IF (PVL.s8098[s8098_mapping.FT_202].PDO.VolumeFlow.Status.eStatus=burkert.eSensor_Status.Low_Low_Alarm)	THEN	tStatus:=ez202_Status.FT202_Low_Low_Flow_Alarm;		END_IF;
IF (PVL.s8098[s8098_mapping.FT_202].PDO.VolumeFlow.Status.eStatus=burkert.eSensor_Status.HiHi_Alarm)	THEN	tStatus:=ez202_Status.FT202_High_High_Flow_Alarm;		END_IF;
IF (PVL.s8098[s8098_mapping.FT_203].PDO.VolumeFlow.Status.eStatus=burkert.eSensor_Status.Low_Low_Alarm)	THEN	tStatus:=ez202_Status.FT203_Low_Low_Flow_Alarm;		END_IF;
IF (PVL.s8098[s8098_mapping.FT_203].PDO.VolumeFlow.Status.eStatus=burkert.eSensor_Status.HiHi_Alarm)	THEN	tStatus:=ez202_Status.FT202_High_High_Flow_Alarm;		END_IF;


IF PVl.s8312[s8312_mapping.PT_202].Status.eStatus= Burkert.eSensor_Status.HiHi_Alarm THEN tStatus:=eZ202_Status.PT202_High_Pressure_Alarm; END_IF;
IF PVl.s8312[s8312_mapping.PT_202].Status.eStatus= Burkert.eSensor_Status.Low_Low_Alarm THEN tStatus:=eZ202_Status.PT202_Low_Pressure_Alarm; END_IF;
///////********		IF PVl.s8312[s8312_mapping.PT_203].Status.eStatus= Burkert.eSensor_Status.HiHi_Alarm THEN tStatus:=eZ202_Status.PT203_High_Pressure_Alarm; END_IF;
///////********		IF PVl.s8312[s8312_mapping.PT_203].Status.eStatus= Burkert.eSensor_Status.Low_Low_Alarm THEN tStatus:=eZ202_Status.PT203_Low_Pressure_Alarm; END_IF;

Test_ALL:=tStatus;
                
END_METHOD

METHOD Test_Drain_P202 : eZ202_Status
  VAR_INPUT
    Status : eZ202_status;
  END_VAR
  VAR
    tStatus : eZ202_Status;
  END_VAR
                  tStatus:=Status;
IF NOT(GVL.Filter_Path_Available) THEN tStatus:=eZ202_Status.No_Filter_Available; END_IF;

//IF NOT(GVL.s3363[s3363_mapping.ACV_203].Ready) 	THEN 	tStatus:=eZ202_Status.ACV203_Not_Ready; 	END_IF;
//IF NOT(GVL.s3363[s3363_mapping.ACV_206].Ready) 	THEN 	tStatus:=eZ202_Status.ACV206_Not_Ready; 	END_IF;
//IF NOT(GVL.s3363[s3363_mapping.ACV_224].Ready) 	THEN 	tStatus:=eZ202_Status.ACV224_Not_Ready; 	END_IF;
//IF NOT(GVL.s3363[s3363_mapping.ACV_225].Ready) 	THEN 	tStatus:=eZ202_Status.ACV225_Not_Ready; 	END_IF;
IF NOT(GVL.s3363[s3363_mapping.ACV_226].Ready) 	THEN 	tStatus:=eZ202_Status.ACV226_Not_Ready; 	END_IF;
IF NOT(Network.VFD[VFD_Mapping.VFD_202].Ready) 	THEN	tStatus:=eZ202_status.P202_Not_Ready;		END_IF;
//IF NOT(Network.VFD[VFD_Mapping.VFD_203].Ready) 	THEN	tStatus:=eZ202_status.P203_Not_Ready;		END_IF;
IF NOT(PVL.Ait[AIT_Mapping.LT_202].Ready) 		THEN	tStatus:=eZ202_Status.LT202_Not_Ready;		END_IF;
//IF NOT(PVL.Ait[AIT_Mapping.LT_202A].Ready) 		THEN	tStatus:=eZ202_Status.LT202A_Not_Ready;		END_IF;
IF NOT(PVl.s8312[s8312_mapping.PT_202].Ready)	THEN	tStatus:=ez202_Status.PT202_Not_Ready;		END_IF;
//IF NOT(PVl.s8312[s8312_mapping.PT_203].Ready)	THEN	tStatus:=ez202_Status.PT203_Not_Ready;		END_IF;
IF NOT(PVL.s8098[s8098_mapping.FT_202].Ready)	THEN	tStatus:=ez202_Status.FT202_Not_Ready;		END_IF;
//IF NOT(PVL.s8098[s8098_mapping.FT_203].Ready)	THEN	tStatus:=ez202_Status.FT203_Not_Ready;		END_IF;
IF gvl.LS[ls_mapping.LSLL_205].Status.eStatus=Burkert.DI_Status.No_Liquid_Detected_Alarm	THEN	tStatus:=eZ202_Status.Drain_Complete;		END_IF;
//IF gvl.LS[ls_mapping.LSLL_203].Status.eStatus=Burkert.DI_Status.No_Liquid_Detected_Alarm	THEN	tStatus:=eZ202_Status.P203_Intake_Empty;		END_IF;
//IF gvl.LS[ls_mapping.LSHH_201].Status.eStatus=Burkert.DI_Status.Liquid_Detected_Alarm		THEN	tStatus:=eZ202_Status.EP101_High_High_Alarm;	END_IF;
//IF (PVL.Ait[AIT_Mapping.LT_202].Ready) 		THEN	tStatus:=eZ202_Status.LT202_Not_Ready;		END_IF;
//IF (PVL.Ait[AIT_Mapping.LT_202A].Ready) 		THEN	tStatus:=eZ202_Status.LT202A_Not_Ready;		END_IF;
//IF GVL.s3363[s3363_mapping.ACV_203].Status.eStatus=Burkert.eACV_Status.Pos_Error THEN	tStatus:=eZ202_Status.ACV203_Error; END_IF;
//IF GVL.s3363[s3363_mapping.ACV_206].Status.eStatus=Burkert.eACV_Status.Pos_Error THEN	tStatus:=eZ202_Status.ACV206_Error; END_IF;
//IF GVL.s3363[s3363_mapping.ACV_224].Status.eStatus=Burkert.eACV_Status.Pos_Error THEN	tStatus:=eZ202_Status.ACV224_Error; END_IF;
//IF GVL.s3363[s3363_mapping.ACV_225].Status.eStatus=Burkert.eACV_Status.Pos_Error THEN	tStatus:=eZ202_Status.ACV225_Error; END_IF;
IF GVL.s3363[s3363_mapping.ACV_226].Status.eStatus=Burkert.eACV_Status.Pos_Error THEN	tStatus:=eZ202_Status.ACV226_Error; END_IF;
//IF PVL.AIT[AIT_Mapping.LT_202].Status.eStatus=Burkert.eSensor_Status.Low_Low_Alarm THEN	tStatus:=eZ202_Status.LT202_Low_Low_Alarm;	END_IF;
//IF PVL.AIT[AIT_Mapping.LT_202A].Status.eStatus=Burkert.eSensor_Status.Low_Low_Alarm THEN	tStatus:=eZ202_Status.LT202A_Low_Low_Alarm;	END_IF;
IF (PVL.s8098[s8098_mapping.FT_202].PDO.VolumeFlow.Status.eStatus=burkert.eSensor_Status.Low_Low_Alarm)	THEN	tStatus:=ez202_Status.FT202_Low_Low_Flow_Alarm;		END_IF;
//IF (PVL.s8098[s8098_mapping.FT_202].PDO.VolumeFlow.Status.eStatus=burkert.eSensor_Status.HiHi_Alarm)	THEN	tStatus:=ez202_Status.FT202_High_High_Flow_Alarm;		END_IF;
//IF (PVL.s8098[s8098_mapping.FT_203].PDO.VolumeFlow.Status.eStatus=burkert.eSensor_Status.Low_Low_Alarm)	THEN	tStatus:=ez202_Status.FT203_Low_Low_Flow_Alarm;		END_IF;
//IF (PVL.s8098[s8098_mapping.FT_203].PDO.VolumeFlow.Status.eStatus=burkert.eSensor_Status.HiHi_Alarm)	THEN	tStatus:=ez202_Status.FT202_High_High_Flow_Alarm;		END_IF;
IF PVl.s8312[s8312_mapping.PT_202].Status.eStatus= Burkert.eSensor_Status.HiHi_Alarm THEN tStatus:=eZ202_Status.PT202_High_Pressure_Alarm; END_IF;
IF PVl.s8312[s8312_mapping.PT_202].Status.eStatus= Burkert.eSensor_Status.Low_Low_Alarm THEN tStatus:=eZ202_Status.PT202_Low_Pressure_Alarm; END_IF;
//IF PVl.s8312[s8312_mapping.PT_203].Status.eStatus= Burkert.eSensor_Status.HiHi_Alarm THEN tStatus:=eZ202_Status.PT203_High_Pressure_Alarm; END_IF;
//IF PVl.s8312[s8312_mapping.PT_203].Status.eStatus= Burkert.eSensor_Status.Low_Low_Alarm THEN tStatus:=eZ202_Status.PT203_Low_Pressure_Alarm; END_IF;

Test_Drain_P202:=tStatus;
                
END_METHOD

METHOD Test_Drain_P203 : eZ202_Status
  VAR_INPUT
    Status : eZ202_status;
  END_VAR
  VAR
    tStatus : eZ202_Status;
  END_VAR
                  tStatus:=Status;
IF NOT(GVL.Filter_Path_Available) THEN tStatus:=eZ202_Status.No_Filter_Available; END_IF;

//IF NOT(GVL.s3363[s3363_mapping.ACV_203].Ready) 	THEN 	tStatus:=eZ202_Status.ACV203_Not_Ready; 	END_IF;
//IF NOT(GVL.s3363[s3363_mapping.ACV_206].Ready) 	THEN 	tStatus:=eZ202_Status.ACV206_Not_Ready; 	END_IF;
//IF NOT(GVL.s3363[s3363_mapping.ACV_224].Ready) 	THEN 	tStatus:=eZ202_Status.ACV224_Not_Ready; 	END_IF;
//IF NOT(GVL.s3363[s3363_mapping.ACV_225].Ready) 	THEN 	tStatus:=eZ202_Status.ACV225_Not_Ready; 	END_IF;
IF NOT(GVL.s3363[s3363_mapping.ACV_226].Ready) 	THEN 	tStatus:=eZ202_Status.ACV226_Not_Ready; 	END_IF;
IF NOT(Network.VFD[VFD_Mapping.VFD_202].Ready) 	THEN	tStatus:=eZ202_status.P202_Not_Ready;		END_IF;
//IF NOT(Network.VFD[VFD_Mapping.VFD_203].Ready) 	THEN	tStatus:=eZ202_status.P203_Not_Ready;		END_IF;
IF NOT(PVL.Ait[AIT_Mapping.LT_202].Ready) 		THEN	tStatus:=eZ202_Status.LT202_Not_Ready;		END_IF;
//IF NOT(PVL.Ait[AIT_Mapping.LT_202A].Ready) 		THEN	tStatus:=eZ202_Status.LT202A_Not_Ready;		END_IF;
IF NOT(PVl.s8312[s8312_mapping.PT_202].Ready)	THEN	tStatus:=ez202_Status.PT202_Not_Ready;		END_IF;
//IF NOT(PVl.s8312[s8312_mapping.PT_203].Ready)	THEN	tStatus:=ez202_Status.PT203_Not_Ready;		END_IF;
IF NOT(PVL.s8098[s8098_mapping.FT_202].Ready)	THEN	tStatus:=ez202_Status.FT202_Not_Ready;		END_IF;
//IF NOT(PVL.s8098[s8098_mapping.FT_203].Ready)	THEN	tStatus:=ez202_Status.FT203_Not_Ready;		END_IF;
//IF gvl.LS[ls_mapping.LSLL_205].Status.eStatus=Burkert.DI_Status.No_Liquid_Detected_Alarm	THEN	tStatus:=eZ202_Status.Drain_Complete;		END_IF;
IF gvl.LS[ls_mapping.LSLL_203].Status.eStatus=Burkert.DI_Status.No_Liquid_Detected_Alarm	THEN	tStatus:=eZ202_Status.Drain_Complete;		END_IF;
//IF gvl.LS[ls_mapping.LSHH_201].Status.eStatus=Burkert.DI_Status.Liquid_Detected_Alarm		THEN	tStatus:=eZ202_Status.EP101_High_High_Alarm;	END_IF;
//IF (PVL.Ait[AIT_Mapping.LT_202].Ready) 		THEN	tStatus:=eZ202_Status.LT202_Not_Ready;		END_IF;
//IF (PVL.Ait[AIT_Mapping.LT_202A].Ready) 		THEN	tStatus:=eZ202_Status.LT202A_Not_Ready;		END_IF;
//IF GVL.s3363[s3363_mapping.ACV_203].Status.eStatus=Burkert.eACV_Status.Pos_Error THEN	tStatus:=eZ202_Status.ACV203_Error; END_IF;
//IF GVL.s3363[s3363_mapping.ACV_206].Status.eStatus=Burkert.eACV_Status.Pos_Error THEN	tStatus:=eZ202_Status.ACV206_Error; END_IF;
//IF GVL.s3363[s3363_mapping.ACV_224].Status.eStatus=Burkert.eACV_Status.Pos_Error THEN	tStatus:=eZ202_Status.ACV224_Error; END_IF;
//IF GVL.s3363[s3363_mapping.ACV_225].Status.eStatus=Burkert.eACV_Status.Pos_Error THEN	tStatus:=eZ202_Status.ACV225_Error; END_IF;
IF GVL.s3363[s3363_mapping.ACV_226].Status.eStatus=Burkert.eACV_Status.Pos_Error THEN	tStatus:=eZ202_Status.ACV226_Error; END_IF;
//IF PVL.AIT[AIT_Mapping.LT_202].Status.eStatus=Burkert.eSensor_Status.Low_Low_Alarm THEN	tStatus:=eZ202_Status.LT202_Low_Low_Alarm;	END_IF;
//IF PVL.AIT[AIT_Mapping.LT_202A].Status.eStatus=Burkert.eSensor_Status.Low_Low_Alarm THEN	tStatus:=eZ202_Status.LT202A_Low_Low_Alarm;	END_IF;
IF (PVL.s8098[s8098_mapping.FT_202].PDO.VolumeFlow.Status.eStatus=burkert.eSensor_Status.Low_Low_Alarm)	THEN	tStatus:=ez202_Status.FT202_Low_Low_Flow_Alarm;		END_IF;
//IF (PVL.s8098[s8098_mapping.FT_202].PDO.VolumeFlow.Status.eStatus=burkert.eSensor_Status.HiHi_Alarm)	THEN	tStatus:=ez202_Status.FT202_High_High_Flow_Alarm;		END_IF;
//IF (PVL.s8098[s8098_mapping.FT_203].PDO.VolumeFlow.Status.eStatus=burkert.eSensor_Status.Low_Low_Alarm)	THEN	tStatus:=ez202_Status.FT203_Low_Low_Flow_Alarm;		END_IF;
//IF (PVL.s8098[s8098_mapping.FT_203].PDO.VolumeFlow.Status.eStatus=burkert.eSensor_Status.HiHi_Alarm)	THEN	tStatus:=ez202_Status.FT202_High_High_Flow_Alarm;		END_IF;
IF PVl.s8312[s8312_mapping.PT_202].Status.eStatus= Burkert.eSensor_Status.HiHi_Alarm THEN tStatus:=eZ202_Status.PT202_High_Pressure_Alarm; END_IF;
IF PVl.s8312[s8312_mapping.PT_202].Status.eStatus= Burkert.eSensor_Status.Low_Low_Alarm THEN tStatus:=eZ202_Status.PT202_Low_Pressure_Alarm; END_IF;
//IF PVl.s8312[s8312_mapping.PT_203].Status.eStatus= Burkert.eSensor_Status.HiHi_Alarm THEN tStatus:=eZ202_Status.PT203_High_Pressure_Alarm; END_IF;
//IF PVl.s8312[s8312_mapping.PT_203].Status.eStatus= Burkert.eSensor_Status.Low_Low_Alarm THEN tStatus:=eZ202_Status.PT203_Low_Pressure_Alarm; END_IF;

Test_Drain_P203:=tStatus;
                
END_METHOD

METHOD Test_Z201_Return_P202 : eZ202_Status
  VAR_INPUT
    Status : eZ202_status;
  END_VAR
  VAR
    tStatus : eZ202_Status;
  END_VAR
                  tStatus:=Status;


IF NOT(GVL.s3363[s3363_mapping.ACV_203].Ready) 	THEN 	tStatus:=eZ202_Status.ACV203_Not_Ready; 	END_IF;
IF NOT(GVL.s3363[s3363_mapping.ACV_206].Ready) 	THEN 	tStatus:=eZ202_Status.ACV206_Not_Ready; 	END_IF;
//IF NOT(GVL.s3363[s3363_mapping.ACV_224].Ready) 	THEN 	tStatus:=eZ202_Status.ACV224_Not_Ready; 	END_IF;
//IF NOT(GVL.s3363[s3363_mapping.ACV_225].Ready) 	THEN 	tStatus:=eZ202_Status.ACV225_Not_Ready; 	END_IF;
IF NOT(GVL.s3363[s3363_mapping.ACV_226].Ready) 	THEN 	tStatus:=eZ202_Status.ACV226_Not_Ready; 	END_IF;

IF NOT(Network.VFD[VFD_Mapping.VFD_202].Ready) 	THEN	tStatus:=eZ202_status.P202_Not_Ready;		END_IF;
//IF NOT(Network.VFD[VFD_Mapping.VFD_203].Ready) 	THEN	tStatus:=eZ202_status.P203_Not_Ready;		END_IF;

IF NOT(PVL.Ait[AIT_Mapping.LT_202].Ready) 		THEN	tStatus:=eZ202_Status.LT202_Not_Ready;		END_IF;
//IF NOT(PVL.Ait[AIT_Mapping.LT_202A].Ready) 		THEN	tStatus:=eZ202_Status.LT202A_Not_Ready;		END_IF;

///////********		IF NOT(PVl.s8312[s8312_mapping.PT_202].Ready)	THEN	tStatus:=ez202_Status.PT202_Not_Ready;		END_IF;
///////********		IF NOT(PVl.s8312[s8312_mapping.PT_203].Ready)	THEN	tStatus:=ez202_Status.PT203_Not_Ready;		END_IF;

//IF NOT(PVL.s8098[s8098_mapping.FT_202].Ready)	THEN	tStatus:=ez202_Status.FT202_Not_Ready;		END_IF;
//IF NOT(PVL.s8098[s8098_mapping.FT_203].Ready)	THEN	tStatus:=ez202_Status.FT203_Not_Ready;		END_IF;
	
IF gvl.LS[ls_mapping.LSLL_205].Status.eStatus=Burkert.DI_Status.No_Liquid_Detected_Alarm	THEN	tStatus:=eZ202_Status.P202_Intake_Empty;		END_IF;
//IF gvl.LS[ls_mapping.LSLL_203].Status.eStatus=Burkert.DI_Status.No_Liquid_Detected_Alarm	THEN	tStatus:=eZ202_Status.P203_Intake_Empty;		END_IF;
IF gvl.LS[ls_mapping.LSHH_201].Status.eStatus=Burkert.DI_Status.Liquid_Detected_Alarm		THEN	tStatus:=eZ202_Status.EP101_High_High_Alarm;	END_IF;

//IF NOT(PVL.Ait[AIT_Mapping.LT_202].Ready) 		THEN	tStatus:=eZ202_Status.LT202_Not_Ready;		END_IF;
//IF (PVL.Ait[AIT_Mapping.LT_202].Status.eStatus=Burkert.eSensor_Status.HiHi_Alarm) 		THEN	tStatus:=eZ202_Status.LT202_High_High_Alarm;		END_IF;

IF NOT(PVL.Ait[AIT_Mapping.LT_201].Ready) 		THEN	tStatus:=eZ202_Status.LT201_Not_Ready;		END_IF;
IF (PVL.Ait[AIT_Mapping.LT_201].Status.eStatus=Burkert.eSensor_Status.HiHi_Alarm) 		THEN	tStatus:=eZ202_Status.LT201_High_High_Alarm;		END_IF;

IF NOT(pVL.Ait[AIT_Mapping.LT_101_P].Ready) 		THEN	tStatus:=eZ202_Status.LT101_Not_Ready;		END_IF;
IF (PVL.Ait[AIT_Mapping.LT_101_P].Status.eStatus=Burkert.eSensor_Status.HiHi_Alarm) 		THEN	tStatus:=eZ202_Status.LT101_High_High_Alarm;		END_IF;

//IF (PVL.Ait[AIT_Mapping.LT_202A].Ready) 		THEN	tStatus:=eZ202_Status.LT202A_Not_Ready;		END_IF;


IF GVL.s3363[s3363_mapping.ACV_203].Status.eStatus=Burkert.eACV_Status.Pos_Error THEN	tStatus:=eZ202_Status.ACV203_Error; END_IF;
IF GVL.s3363[s3363_mapping.ACV_206].Status.eStatus=Burkert.eACV_Status.Pos_Error THEN	tStatus:=eZ202_Status.ACV206_Error; END_IF;
//IF GVL.s3363[s3363_mapping.ACV_224].Status.eStatus=Burkert.eACV_Status.Pos_Error THEN	tStatus:=eZ202_Status.ACV224_Error; END_IF;
//IF GVL.s3363[s3363_mapping.ACV_225].Status.eStatus=Burkert.eACV_Status.Pos_Error THEN	tStatus:=eZ202_Status.ACV225_Error; END_IF;
IF GVL.s3363[s3363_mapping.ACV_226].Status.eStatus=Burkert.eACV_Status.Pos_Error THEN	tStatus:=eZ202_Status.ACV226_Error; END_IF;

//IF NOT(GVL.Filter_Path_Available) THEN tStatus:=eZ202_Status.No_Filter_Available; END_IF;

//IF (PVL.s8098[s8098_mapping.FT_202].PDO.VolumeFlow.Status.eStatus=burkert.eSensor_Status.Low_Low_Alarm)	THEN	tStatus:=ez202_Status.FT202_Low_Low_Flow_Alarm;		END_IF;
//IF (PVL.s8098[s8098_mapping.FT_202].PDO.VolumeFlow.Status.eStatus=burkert.eSensor_Status.HiHi_Alarm)	THEN	tStatus:=ez202_Status.FT202_High_High_Flow_Alarm;		END_IF;
IF (PVL.s8098[s8098_mapping.FT_203].PDO.VolumeFlow.Status.eStatus=burkert.eSensor_Status.Low_Low_Alarm)	THEN	tStatus:=ez202_Status.FT203_Low_Low_Flow_Alarm;		END_IF;
//IF (PVL.s8098[s8098_mapping.FT_203].PDO.VolumeFlow.Status.eStatus=burkert.eSensor_Status.HiHi_Alarm)	THEN	tStatus:=ez202_Status.FT202_High_High_Flow_Alarm;		END_IF;


//IF PVl.s8312[s8312_mapping.PT_202].Status.eStatus= Burkert.eSensor_Status.HiHi_Alarm THEN tStatus:=eZ202_Status.PT202_High_Pressure_Alarm; END_IF;
//IF PVl.s8312[s8312_mapping.PT_202].Status.eStatus= Burkert.eSensor_Status.Low_Low_Alarm THEN tStatus:=eZ202_Status.PT202_Low_Pressure_Alarm; END_IF;
///////********		IF PVl.s8312[s8312_mapping.PT_203].Status.eStatus= Burkert.eSensor_Status.HiHi_Alarm THEN tStatus:=eZ202_Status.PT203_High_Pressure_Alarm; END_IF;
///////********		IF PVl.s8312[s8312_mapping.PT_203].Status.eStatus= Burkert.eSensor_Status.Low_Low_Alarm THEN tStatus:=eZ202_Status.PT203_Low_Pressure_Alarm; END_IF;

IF (PVL.Ait[AIT_Mapping.LT_202].Status.eStatus=Burkert.eSensor_Status.Low_Low_Alarm) 		THEN	tStatus:=eZ202_Status.LT202_Low_Low_Alarm;		END_IF;

Test_Z201_Return_P202:=tStatus;
                
END_METHOD

METHOD Test_Z201_Return_P203 : eZ202_Status
  VAR_INPUT
    Status : eZ202_status;
  END_VAR
  VAR
    tStatus : eZ202_Status;
  END_VAR
                  tStatus:=Status;


IF NOT(GVL.s3363[s3363_mapping.ACV_203].Ready) 	THEN 	tStatus:=eZ202_Status.ACV203_Not_Ready; 	END_IF;
//IF NOT(GVL.s3363[s3363_mapping.ACV_206].Ready) 	THEN 	tStatus:=eZ202_Status.ACV206_Not_Ready; 	END_IF;
//IF NOT(GVL.s3363[s3363_mapping.ACV_224].Ready) 	THEN 	tStatus:=eZ202_Status.ACV224_Not_Ready; 	END_IF;
//IF NOT(GVL.s3363[s3363_mapping.ACV_225].Ready) 	THEN 	tStatus:=eZ202_Status.ACV225_Not_Ready; 	END_IF;
IF NOT(GVL.s3363[s3363_mapping.ACV_226].Ready) 	THEN 	tStatus:=eZ202_Status.ACV226_Not_Ready; 	END_IF;

//IF NOT(Network.VFD[VFD_Mapping.VFD_202].Ready) 	THEN	tStatus:=eZ202_status.P202_Not_Ready;		END_IF;
IF NOT(Network.VFD[VFD_Mapping.VFD_203].Ready) 	THEN	tStatus:=eZ202_status.P203_Not_Ready;		END_IF;

IF NOT(PVL.Ait[AIT_Mapping.LT_202].Ready) 		THEN	tStatus:=eZ202_Status.LT202_Not_Ready;		END_IF;
//IF NOT(PVL.Ait[AIT_Mapping.LT_202A].Ready) 		THEN	tStatus:=eZ202_Status.LT202A_Not_Ready;		END_IF;

//IF NOT(PVl.s8312[s8312_mapping.PT_202].Ready)	THEN	tStatus:=ez202_Status.PT202_Not_Ready;		END_IF;
///////********		IF NOT(PVl.s8312[s8312_mapping.PT_203].Ready)	THEN	tStatus:=ez202_Status.PT203_Not_Ready;		END_IF;

//IF NOT(PVL.s8098[s8098_mapping.FT_202].Ready)	THEN	tStatus:=ez202_Status.FT202_Not_Ready;		END_IF;
//IF NOT(PVL.s8098[s8098_mapping.FT_203].Ready)	THEN	tStatus:=ez202_Status.FT203_Not_Ready;		END_IF;
	
//IF gvl.LS[ls_mapping.LSLL_205].Status.eStatus=Burkert.DI_Status.No_Liquid_Detected_Alarm	THEN	tStatus:=eZ202_Status.P202_Intake_Empty;		END_IF;
IF gvl.LS[ls_mapping.LSLL_203].Status.eStatus=Burkert.DI_Status.No_Liquid_Detected_Alarm	THEN	tStatus:=eZ202_Status.P203_Intake_Empty;		END_IF;
IF gvl.LS[ls_mapping.LSHH_201].Status.eStatus=Burkert.DI_Status.Liquid_Detected_Alarm		THEN	tStatus:=eZ202_Status.EP101_High_High_Alarm;	END_IF;

//IF NOT(PVL.Ait[AIT_Mapping.LT_202].Ready) 		THEN	tStatus:=eZ202_Status.LT202_Not_Ready;		END_IF;
//IF (PVL.Ait[AIT_Mapping.LT_202].Status.eStatus=Burkert.eSensor_Status.HiHi_Alarm) 		THEN	tStatus:=eZ202_Status.LT202_High_High_Alarm;		END_IF;

IF NOT(PVL.Ait[AIT_Mapping.LT_201].Ready) 		THEN	tStatus:=eZ202_Status.LT201_Not_Ready;		END_IF;
IF (PVL.Ait[AIT_Mapping.LT_201].Status.eStatus=Burkert.eSensor_Status.HiHi_Alarm) 		THEN	tStatus:=eZ202_Status.LT201_High_High_Alarm;		END_IF;

IF NOT(PVL.Ait[AIT_Mapping.LT_101_p].Ready) 		THEN	tStatus:=eZ202_Status.LT101_Not_Ready;		END_IF;
IF (PVL.Ait[AIT_Mapping.LT_101_P].Status.eStatus=Burkert.eSensor_Status.HiHi_Alarm) 		THEN	tStatus:=eZ202_Status.LT101_High_High_Alarm;		END_IF;


IF GVL.s3363[s3363_mapping.ACV_203].Status.eStatus=Burkert.eACV_Status.Pos_Error THEN	tStatus:=eZ202_Status.ACV203_Error; END_IF;
//IF GVL.s3363[s3363_mapping.ACV_206].Status.eStatus=Burkert.eACV_Status.Pos_Error THEN	tStatus:=eZ202_Status.ACV206_Error; END_IF;
//IF GVL.s3363[s3363_mapping.ACV_224].Status.eStatus=Burkert.eACV_Status.Pos_Error THEN	tStatus:=eZ202_Status.ACV224_Error; END_IF;
//IF GVL.s3363[s3363_mapping.ACV_225].Status.eStatus=Burkert.eACV_Status.Pos_Error THEN	tStatus:=eZ202_Status.ACV225_Error; END_IF;
IF GVL.s3363[s3363_mapping.ACV_226].Status.eStatus=Burkert.eACV_Status.Pos_Error THEN	tStatus:=eZ202_Status.ACV226_Error; END_IF;

//IF NOT(GVL.Filter_Path_Available) THEN tStatus:=eZ202_Status.No_Filter_Available; END_IF;

//IF (PVL.s8098[s8098_mapping.FT_202].PDO.VolumeFlow.Status.eStatus=burkert.eSensor_Status.Low_Low_Alarm)	THEN	tStatus:=ez202_Status.FT202_Low_Low_Flow_Alarm;		END_IF;
//IF (PVL.s8098[s8098_mapping.FT_202].PDO.VolumeFlow.Status.eStatus=burkert.eSensor_Status.HiHi_Alarm)	THEN	tStatus:=ez202_Status.FT202_High_High_Flow_Alarm;		END_IF;
IF (PVL.s8098[s8098_mapping.FT_203].PDO.VolumeFlow.Status.eStatus=burkert.eSensor_Status.Low_Low_Alarm)	THEN	tStatus:=ez202_Status.FT203_Low_Low_Flow_Alarm;		END_IF;
//IF (PVL.s8098[s8098_mapping.FT_203].PDO.VolumeFlow.Status.eStatus=burkert.eSensor_Status.HiHi_Alarm)	THEN	tStatus:=ez202_Status.FT202_High_High_Flow_Alarm;		END_IF;


//IF PVl.s8312[s8312_mapping.PT_202].Status.eStatus= Burkert.eSensor_Status.HiHi_Alarm THEN tStatus:=eZ202_Status.PT202_High_Pressure_Alarm; END_IF;
//IF PVl.s8312[s8312_mapping.PT_202].Status.eStatus= Burkert.eSensor_Status.Low_Low_Alarm THEN tStatus:=eZ202_Status.PT202_Low_Pressure_Alarm; END_IF;
///////********		IF PVl.s8312[s8312_mapping.PT_203].Status.eStatus= Burkert.eSensor_Status.HiHi_Alarm THEN tStatus:=eZ202_Status.PT203_High_Pressure_Alarm; END_IF;
///////********		IF PVl.s8312[s8312_mapping.PT_203].Status.eStatus= Burkert.eSensor_Status.Low_Low_Alarm THEN tStatus:=eZ202_Status.PT203_Low_Pressure_Alarm; END_IF;


IF (PVL.Ait[AIT_Mapping.LT_202].Status.eStatus=Burkert.eSensor_Status.Low_Low_Alarm) 		THEN	tStatus:=eZ202_Status.LT202_Low_Low_Alarm;		END_IF;
Test_Z201_Return_p203:=tStatus;
                
END_METHOD

METHOD Test_Filters_P203 : eZ202_Status
  VAR_INPUT
    Status : eZ202_status;
  END_VAR
  VAR
    tStatus : eZ202_Status;
  END_VAR
                  tStatus:=Status;
IF NOT(GVL.Filter_Path_Available) THEN tStatus:=eZ202_Status.No_Filter_Available; END_IF;


//IF NOT(GVL.s3363[s3363_mapping.ACV_203].Ready) 	THEN 	tStatus:=eZ202_Status.ACV203_Not_Ready; 	END_IF;
IF NOT(GVL.s3363[s3363_mapping.ACV_206].Ready) 	THEN 	tStatus:=eZ202_Status.ACV206_Not_Ready; 	END_IF;
//IF NOT(GVL.s3363[s3363_mapping.ACV_224].Ready) 	THEN 	tStatus:=eZ202_Status.ACV224_Not_Ready; 	END_IF;
//IF NOT(GVL.s3363[s3363_mapping.ACV_225].Ready) 	THEN 	tStatus:=eZ202_Status.ACV225_Not_Ready; 	END_IF;
IF NOT(GVL.s3363[s3363_mapping.ACV_226].Ready) 	THEN 	tStatus:=eZ202_Status.ACV226_Not_Ready; 	END_IF;

//IF NOT(Network.VFD[VFD_Mapping.VFD_202].Ready) 	THEN	tStatus:=eZ202_status.P202_Not_Ready;		END_IF;
IF NOT(Network.VFD[VFD_Mapping.VFD_203].Ready) 	THEN	tStatus:=eZ202_status.P203_Not_Ready;		END_IF;

IF NOT(PVL.Ait[AIT_Mapping.LT_202].Ready) 		THEN	tStatus:=eZ202_Status.LT202_Not_Ready;		END_IF;
//IF NOT(PVL.Ait[AIT_Mapping.LT_202A].Ready) 		THEN	tStatus:=eZ202_Status.LT202A_Not_Ready;		END_IF;

//IF NOT(PVl.s8312[s8312_mapping.PT_202].Ready)	THEN	tStatus:=ez202_Status.PT202_Not_Ready;		END_IF;
IF NOT(PVl.s8312[s8312_mapping.PT_203].Ready)	THEN	tStatus:=ez202_Status.PT203_Not_Ready;		END_IF;

IF NOT(PVL.s8098[s8098_mapping.FT_202].Ready)	THEN	tStatus:=ez202_Status.FT202_Not_Ready;		END_IF;
//IF NOT(PVL.s8098[s8098_mapping.FT_203].Ready)	THEN	tStatus:=ez202_Status.FT203_Not_Ready;		END_IF;
	
//IF gvl.LS[ls_mapping.LSLL_205].Status.eStatus=Burkert.DI_Status.No_Liquid_Detected_Alarm	THEN	tStatus:=eZ202_Status.P202_Intake_Empty;		END_IF;
IF gvl.LS[ls_mapping.LSLL_203].Status.eStatus=Burkert.DI_Status.No_Liquid_Detected_Alarm	THEN	tStatus:=eZ202_Status.P203_Intake_Empty;		END_IF;
//IF gvl.LS[ls_mapping.LSHH_201].Status.eStatus=Burkert.DI_Status.Liquid_Detected_Alarm		THEN	tStatus:=eZ202_Status.EP101_High_High_Alarm;	END_IF;




//IF GVL.s3363[s3363_mapping.ACV_203].Status.eStatus=Burkert.eACV_Status.Pos_Error THEN	tStatus:=eZ202_Status.ACV203_Error; END_IF;
IF GVL.s3363[s3363_mapping.ACV_206].Status.eStatus=Burkert.eACV_Status.Pos_Error THEN	tStatus:=eZ202_Status.ACV206_Error; END_IF;
//IF GVL.s3363[s3363_mapping.ACV_224].Status.eStatus=Burkert.eACV_Status.Pos_Error THEN	tStatus:=eZ202_Status.ACV224_Error; END_IF;
//IF GVL.s3363[s3363_mapping.ACV_225].Status.eStatus=Burkert.eACV_Status.Pos_Error THEN	tStatus:=eZ202_Status.ACV225_Error; END_IF;
IF GVL.s3363[s3363_mapping.ACV_226].Status.eStatus=Burkert.eACV_Status.Pos_Error THEN	tStatus:=eZ202_Status.ACV226_Error; END_IF;



IF PVL.AIT[AIT_Mapping.LT_202].Status.eStatus=Burkert.eSensor_Status.Low_Low_Alarm THEN	tStatus:=eZ202_Status.LT202_Low_Low_Alarm;	END_IF;

//IF PVL.AIT[AIT_Mapping.LT_202A].Status.eStatus=Burkert.eSensor_Status.Low_Low_Alarm THEN	tStatus:=eZ202_Status.LT202A_Low_Low_Alarm;	END_IF;

IF (PVL.s8098[s8098_mapping.FT_202].PDO.VolumeFlow.Status.eStatus=burkert.eSensor_Status.Low_Low_Alarm)	THEN	tStatus:=ez202_Status.FT202_Low_Low_Flow_Alarm;		END_IF;
//IF (PVL.s8098[s8098_mapping.FT_202].PDO.VolumeFlow.Status.eStatus=burkert.eSensor_Status.HiHi_Alarm)	THEN	tStatus:=ez202_Status.FT202_High_High_Flow_Alarm;		END_IF;
//IF NOT(PVL.s8098[s8098_mapping.FT_203].PDO.VolumeFlow.Status.eStatus=burkert.eSensor_Status.Low_Low_Alarm)	THEN	tStatus:=ez202_Status.FT203_Low_Low_Flow_Alarm;		END_IF;
//IF NOT(PVL.s8098[s8098_mapping.FT_203].PDO.VolumeFlow.Status.eStatus=burkert.eSensor_Status.HiHi_Alarm)	THEN	tStatus:=ez202_Status.FT202_High_High_Flow_Alarm;		END_IF;
IF (PVL.s8098[s8098_mapping.FT_202].PDO.VolumeFlow.Status.eStatus=burkert.eSensor_Status.Low_Low_Alarm)	THEN	tStatus:=ez202_Status.FT202_Low_Low_Flow_Alarm;		END_IF;
//IF (PVL.s8098[s8098_mapping.FT_202].PDO.VolumeFlow.Status.eStatus=burkert.eSensor_Status.HiHi_Alarm)	THEN	tStatus:=ez202_Status.FT202_High_High_Flow_Alarm;		END_IF;
//IF (PVL.s8098[s8098_mapping.FT_203].PDO.VolumeFlow.Status.eStatus=burkert.eSensor_Status.Low_Low_Alarm)	THEN	tStatus:=ez202_Status.FT203_Low_Low_Flow_Alarm;		END_IF;
//IF (PVL.s8098[s8098_mapping.FT_203].PDO.VolumeFlow.Status.eStatus=burkert.eSensor_Status.HiHi_Alarm)	THEN	tStatus:=ez202_Status.FT202_High_High_Flow_Alarm;		END_IF;


IF PVl.s8312[s8312_mapping.PT_202].Status.eStatus= Burkert.eSensor_Status.HiHi_Alarm THEN tStatus:=eZ202_Status.PT202_High_Pressure_Alarm; END_IF;
IF PVl.s8312[s8312_mapping.PT_202].Status.eStatus= Burkert.eSensor_Status.Low_Low_Alarm THEN tStatus:=eZ202_Status.PT202_Low_Pressure_Alarm; END_IF;
//IF PVl.s8312[s8312_mapping.PT_203].Status.eStatus= Burkert.eSensor_Status.HiHi_Alarm THEN tStatus:=eZ202_Status.PT203_High_Pressure_Alarm; END_IF;
//IF PVl.s8312[s8312_mapping.PT_203].Status.eStatus= Burkert.eSensor_Status.Low_Low_Alarm THEN tStatus:=eZ202_Status.PT203_Low_Pressure_Alarm; END_IF;

Test_Filters_P203:=tStatus;




                
END_METHOD

METHOD Test_Combined_Level : eZ202_Status
  VAR_INPUT
    Status : eZ202_status;
  END_VAR
  VAR
    tStatus : eZ202_Status;
  END_VAR
                  tStatus:=Status;


IF NOT(GVL.s3363[s3363_mapping.ACV_203].Ready) 	THEN 	tStatus:=eZ202_Status.ACV203_Not_Ready; 	END_IF;
IF NOT(GVL.s3363[s3363_mapping.ACV_206].Ready) 	THEN 	tStatus:=eZ202_Status.ACV206_Not_Ready; 	END_IF;
//IF NOT(GVL.s3363[s3363_mapping.ACV_224].Ready) 	THEN 	tStatus:=eZ202_Status.ACV224_Not_Ready; 	END_IF;
//IF NOT(GVL.s3363[s3363_mapping.ACV_225].Ready) 	THEN 	tStatus:=eZ202_Status.ACV225_Not_Ready; 	END_IF;
IF NOT(GVL.s3363[s3363_mapping.ACV_226].Ready) 	THEN 	tStatus:=eZ202_Status.ACV226_Not_Ready; 	END_IF;

IF NOT(Network.VFD[VFD_Mapping.VFD_202].Ready) 	THEN	tStatus:=eZ202_status.P202_Not_Ready;		END_IF;
IF NOT(Network.VFD[VFD_Mapping.VFD_203].Ready) 	THEN	tStatus:=eZ202_status.P203_Not_Ready;		END_IF;

IF NOT(PVL.Ait[AIT_Mapping.LT_202].Ready) 		THEN	tStatus:=eZ202_Status.LT202_Not_Ready;		END_IF;
IF NOT(PVL.Ait[AIT_Mapping.LT_202A].Ready) 		THEN	tStatus:=eZ202_Status.LT202A_Not_Ready;		END_IF;

IF (PVL.Ait[AIT_Mapping.LT_202].Ready) 		THEN	tStatus:=eZ202_Status.LT202_Not_Ready;		END_IF;
IF (PVL.Ait[AIT_Mapping.LT_202].Status.eStatus=Burkert.eSensor_Status.HiHi_Alarm) 		THEN	tStatus:=eZ202_Status.LT202_High_High_Alarm;		END_IF;

IF (PVL.Ait[AIT_Mapping.LT_201].Ready) 		THEN	tStatus:=eZ202_Status.LT201_Not_Ready;		END_IF;
IF (PVL.Ait[AIT_Mapping.LT_201].Status.eStatus=Burkert.eSensor_Status.HiHi_Alarm) 		THEN	tStatus:=eZ202_Status.LT201_High_High_Alarm;		END_IF;

IF (PVL.Ait[AIT_Mapping.LT_101_p].Ready) 		THEN	tStatus:=eZ202_Status.LT101_Not_Ready;		END_IF;
IF (PVL.Ait[AIT_Mapping.LT_101_P].Status.eStatus=Burkert.eSensor_Status.HiHi_Alarm) 		THEN	tStatus:=eZ202_Status.LT101_High_High_Alarm;		END_IF;

IF NOT(PVl.s8312[s8312_mapping.PT_202].Ready)	THEN	tStatus:=ez202_Status.PT202_Not_Ready;		END_IF;
///////********		IF NOT(PVl.s8312[s8312_mapping.PT_203].Ready)	THEN	tStatus:=ez202_Status.PT203_Not_Ready;		END_IF;

IF NOT(PVL.s8098[s8098_mapping.FT_202].Ready)	THEN	tStatus:=ez202_Status.FT202_Not_Ready;		END_IF;
//IF NOT(PVL.s8098[s8098_mapping.FT_203].Ready)	THEN	tStatus:=ez202_Status.FT203_Not_Ready;		END_IF;
	
IF gvl.LS[ls_mapping.LSLL_205].Status.eStatus=Burkert.DI_Status.No_Liquid_Detected_Alarm	THEN	tStatus:=eZ202_Status.P202_Intake_Empty;		END_IF;
IF gvl.LS[ls_mapping.LSLL_203].Status.eStatus=Burkert.DI_Status.No_Liquid_Detected_Alarm	THEN	tStatus:=eZ202_Status.P203_Intake_Empty;		END_IF;
IF gvl.LS[ls_mapping.LSHH_201].Status.eStatus=Burkert.DI_Status.Liquid_Detected_Alarm		THEN	tStatus:=eZ202_Status.EP101_High_High_Alarm;	END_IF;

//IF (PVL.Ait[AIT_Mapping.LT_202].Ready) 		THEN	tStatus:=eZ202_Status.LT202_Not_Ready;		END_IF;
//IF (PVL.Ait[AIT_Mapping.LT_202A].Ready) 		THEN	tStatus:=eZ202_Status.LT202A_Not_Ready;		END_IF;


IF GVL.s3363[s3363_mapping.ACV_203].Status.eStatus=Burkert.eACV_Status.Pos_Error THEN	tStatus:=eZ202_Status.ACV203_Error; END_IF;
IF GVL.s3363[s3363_mapping.ACV_206].Status.eStatus=Burkert.eACV_Status.Pos_Error THEN	tStatus:=eZ202_Status.ACV206_Error; END_IF;
//IF GVL.s3363[s3363_mapping.ACV_224].Status.eStatus=Burkert.eACV_Status.Pos_Error THEN	tStatus:=eZ202_Status.ACV224_Error; END_IF;
//IF GVL.s3363[s3363_mapping.ACV_225].Status.eStatus=Burkert.eACV_Status.Pos_Error THEN	tStatus:=eZ202_Status.ACV225_Error; END_IF;
IF GVL.s3363[s3363_mapping.ACV_226].Status.eStatus=Burkert.eACV_Status.Pos_Error THEN	tStatus:=eZ202_Status.ACV226_Error; END_IF;


//IF NOT(GVL.Filter_Path_Available) THEN tStatus:=eZ202_Status.No_Filter_Available; END_IF;


/////////////////////////////
	

IF NOT(GVL.Filter_Path_Available) THEN tStatus:=eZ202_Status.No_Filter_Available; END_IF;

IF PVL.AIT[AIT_Mapping.LT_202].Status.eStatus=Burkert.eSensor_Status.Low_Low_Alarm THEN	tStatus:=eZ202_Status.LT202_Low_Low_Alarm;	END_IF;
//IF PVL.AIT[AIT_Mapping.LT_202A].Status.eStatus=Burkert.eSensor_Status.Low_Low_Alarm THEN	tStatus:=eZ202_Status.LT202A_Low_Low_Alarm;	END_IF;

//IF (PVL.s8098[s8098_mapping.FT_202].PDO.VolumeFlow.Status.eStatus=burkert.eSensor_Status.Low_Low_Alarm)	THEN	tStatus:=ez202_Status.FT202_Low_Low_Flow_Alarm;		END_IF;
//IF (PVL.s8098[s8098_mapping.FT_202].PDO.VolumeFlow.Status.eStatus=burkert.eSensor_Status.HiHi_Alarm)	THEN	tStatus:=ez202_Status.FT202_High_High_Flow_Alarm;		END_IF;
//IF (PVL.s8098[s8098_mapping.FT_203].PDO.VolumeFlow.Status.eStatus=burkert.eSensor_Status.Low_Low_Alarm)	THEN	tStatus:=ez202_Status.FT203_Low_Low_Flow_Alarm;		END_IF;
//IF (PVL.s8098[s8098_mapping.FT_203].PDO.VolumeFlow.Status.eStatus=burkert.eSensor_Status.HiHi_Alarm)	THEN	tStatus:=ez202_Status.FT202_High_High_Flow_Alarm;		END_IF;


IF PVl.s8312[s8312_mapping.PT_202].Status.eStatus= Burkert.eSensor_Status.HiHi_Alarm THEN tStatus:=eZ202_Status.PT202_High_Pressure_Alarm; END_IF;
IF PVl.s8312[s8312_mapping.PT_202].Status.eStatus= Burkert.eSensor_Status.Low_Low_Alarm THEN tStatus:=eZ202_Status.PT202_Low_Pressure_Alarm; END_IF;
///////********		IF PVl.s8312[s8312_mapping.PT_203].Status.eStatus= Burkert.eSensor_Status.HiHi_Alarm THEN tStatus:=eZ202_Status.PT203_High_Pressure_Alarm; END_IF;
///////********		IF PVl.s8312[s8312_mapping.PT_203].Status.eStatus= Burkert.eSensor_Status.Low_Low_Alarm THEN tStatus:=eZ202_Status.PT203_Low_Pressure_Alarm; END_IF;

IF NOT(PVL.Ait[AIT_Mapping.LT_202].Ready) 		THEN	tStatus:=eZ202_Status.LT202_Not_Ready;		END_IF;
IF (PVL.Ait[AIT_Mapping.LT_202].Status.eStatus=Burkert.eSensor_Status.HiHi_Alarm) 		THEN	tStatus:=eZ202_Status.LT202_High_High_Alarm;		END_IF;

IF NOT(PVL.Ait[AIT_Mapping.LT_201].Ready) 		THEN	tStatus:=eZ202_Status.LT201_Not_Ready;		END_IF;
IF (PVL.Ait[AIT_Mapping.LT_201].Status.eStatus=Burkert.eSensor_Status.HiHi_Alarm) 		THEN	tStatus:=eZ202_Status.LT201_High_High_Alarm;		END_IF;

IF NOT(PVL.Ait[AIT_Mapping.LT_101_p].Ready) 		THEN	tStatus:=eZ202_Status.LT101_Not_Ready;		END_IF;
IF (PVL.Ait[AIT_Mapping.LT_101_P].Status.eStatus=Burkert.eSensor_Status.HiHi_Alarm) 		THEN	tStatus:=eZ202_Status.LT101_High_High_Alarm;		END_IF;

IF (PVL.Ait[AIT_Mapping.LT_202].Status.eStatus=Burkert.eSensor_Status.Low_Low_Alarm) 		THEN	tStatus:=eZ202_Status.LT202_Low_Low_Alarm;		END_IF;





Test_Combined_Level:=tStatus;
                
END_METHOD

METHOD Test_Filters_P202_Level : eZ202_Status
  VAR_INPUT
    Status : eZ202_status;
  END_VAR
  VAR
    tStatus : eZ202_Status;
  END_VAR
                  tStatus:=Status;
IF NOT(GVL.Filter_Path_Available) THEN tStatus:=eZ202_Status.No_Filter_Available; END_IF;


//IF NOT(GVL.s3363[s3363_mapping.ACV_203].Ready) 	THEN 	tStatus:=eZ202_Status.ACV203_Not_Ready; 	END_IF;
//IF NOT(GVL.s3363[s3363_mapping.ACV_206].Ready) 	THEN 	tStatus:=eZ202_Status.ACV206_Not_Ready; 	END_IF;
//IF NOT(GVL.s3363[s3363_mapping.ACV_224].Ready) 	THEN 	tStatus:=eZ202_Status.ACV224_Not_Ready; 	END_IF;
//IF NOT(GVL.s3363[s3363_mapping.ACV_225].Ready) 	THEN 	tStatus:=eZ202_Status.ACV225_Not_Ready; 	END_IF;
IF NOT(GVL.s3363[s3363_mapping.ACV_226].Ready) 	THEN 	tStatus:=eZ202_Status.ACV226_Not_Ready; 	END_IF;

IF NOT(Network.VFD[VFD_Mapping.VFD_202].Ready) 	THEN	tStatus:=eZ202_status.P202_Not_Ready;		END_IF;
//IF NOT(Network.VFD[VFD_Mapping.VFD_203].Ready) 	THEN	tStatus:=eZ202_status.P203_Not_Ready;		END_IF;

IF NOT(PVL.Ait[AIT_Mapping.LT_202].Ready) 		THEN	tStatus:=eZ202_Status.LT202_Not_Ready;		END_IF;
//IF NOT(PVL.Ait[AIT_Mapping.LT_202A].Ready) 		THEN	tStatus:=eZ202_Status.LT202A_Not_Ready;		END_IF;

IF NOT(PVl.s8312[s8312_mapping.PT_202].Ready)	THEN	tStatus:=ez202_Status.PT202_Not_Ready;		END_IF;
//IF NOT(PVl.s8312[s8312_mapping.PT_203].Ready)	THEN	tStatus:=ez202_Status.PT203_Not_Ready;		END_IF;

IF NOT(PVL.s8098[s8098_mapping.FT_202].Ready)	THEN	tStatus:=ez202_Status.FT202_Not_Ready;		END_IF;
//IF NOT(PVL.s8098[s8098_mapping.FT_203].Ready)	THEN	tStatus:=ez202_Status.FT203_Not_Ready;		END_IF;
	
IF gvl.LS[ls_mapping.LSLL_205].Status.eStatus=Burkert.DI_Status.No_Liquid_Detected_Alarm	THEN	tStatus:=eZ202_Status.P202_Intake_Empty;		END_IF;
//IF gvl.LS[ls_mapping.LSLL_203].Status.eStatus=Burkert.DI_Status.No_Liquid_Detected_Alarm	THEN	tStatus:=eZ202_Status.P203_Intake_Empty;		END_IF;
//IF gvl.LS[ls_mapping.LSHH_201].Status.eStatus=Burkert.DI_Status.Liquid_Detected_Alarm		THEN	tStatus:=eZ202_Status.EP101_High_High_Alarm;	END_IF;




//IF GVL.s3363[s3363_mapping.ACV_203].Status.eStatus=Burkert.eACV_Status.Pos_Error THEN	tStatus:=eZ202_Status.ACV203_Error; END_IF;
//IF GVL.s3363[s3363_mapping.ACV_206].Status.eStatus=Burkert.eACV_Status.Pos_Error THEN	tStatus:=eZ202_Status.ACV206_Error; END_IF;
//IF GVL.s3363[s3363_mapping.ACV_224].Status.eStatus=Burkert.eACV_Status.Pos_Error THEN	tStatus:=eZ202_Status.ACV224_Error; END_IF;
//IF GVL.s3363[s3363_mapping.ACV_225].Status.eStatus=Burkert.eACV_Status.Pos_Error THEN	tStatus:=eZ202_Status.ACV225_Error; END_IF;
IF GVL.s3363[s3363_mapping.ACV_226].Status.eStatus=Burkert.eACV_Status.Pos_Error THEN	tStatus:=eZ202_Status.ACV226_Error; END_IF;


IF PVL.AIT[AIT_Mapping.LT_202].Status.eStatus=Burkert.eSensor_Status.Low_Low_Alarm THEN	tStatus:=eZ202_Status.LT202_Low_Low_Alarm;	END_IF;
//IF PVL.AIT[AIT_Mapping.LT_202A].Status.eStatus=Burkert.eSensor_Status.Low_Low_Alarm THEN	tStatus:=eZ202_Status.LT202A_Low_Low_Alarm;	END_IF;

//IF (PVL.s8098[s8098_mapping.FT_202].PDO.VolumeFlow.Status.eStatus=burkert.eSensor_Status.Low_Low_Alarm)	THEN	tStatus:=ez202_Status.FT202_Low_Low_Flow_Alarm;		END_IF;
//IF NOT(PVL.s8098[s8098_mapping.FT_202].PDO.VolumeFlow.Status.eStatus=burkert.eSensor_Status.HiHi_Alarm)	THEN	tStatus:=ez202_Status.FT202_High_High_Flow_Alarm;		END_IF;
//IF NOT(PVL.s8098[s8098_mapping.FT_203].PDO.VolumeFlow.Status.eStatus=burkert.eSensor_Status.Low_Low_Alarm)	THEN	tStatus:=ez202_Status.FT203_Low_Low_Flow_Alarm;		END_IF;
//IF NOT(PVL.s8098[s8098_mapping.FT_203].PDO.VolumeFlow.Status.eStatus=burkert.eSensor_Status.HiHi_Alarm)	THEN	tStatus:=ez202_Status.FT202_High_High_Flow_Alarm;		END_IF;

//IF (PVL.s8098[s8098_mapping.FT_202].PDO.VolumeFlow.Status.eStatus=burkert.eSensor_Status.Low_Low_Alarm)	THEN	tStatus:=ez202_Status.FT202_Low_Low_Flow_Alarm;		END_IF;
//IF (PVL.s8098[s8098_mapping.FT_202].PDO.VolumeFlow.Status.eStatus=burkert.eSensor_Status.HiHi_Alarm)	THEN	tStatus:=ez202_Status.FT202_High_High_Flow_Alarm;		END_IF;
//IF (PVL.s8098[s8098_mapping.FT_203].PDO.VolumeFlow.Status.eStatus=burkert.eSensor_Status.Low_Low_Alarm)	THEN	tStatus:=ez202_Status.FT203_Low_Low_Flow_Alarm;		END_IF;
//IF (PVL.s8098[s8098_mapping.FT_203].PDO.VolumeFlow.Status.eStatus=burkert.eSensor_Status.HiHi_Alarm)	THEN	tStatus:=ez202_Status.FT202_High_High_Flow_Alarm;		END_IF;


IF PVl.s8312[s8312_mapping.PT_202].Status.eStatus= Burkert.eSensor_Status.HiHi_Alarm THEN tStatus:=eZ202_Status.PT202_High_Pressure_Alarm; END_IF;
IF PVl.s8312[s8312_mapping.PT_202].Status.eStatus= Burkert.eSensor_Status.Low_Low_Alarm THEN tStatus:=eZ202_Status.PT202_Low_Pressure_Alarm; END_IF;
//IF PVl.s8312[s8312_mapping.PT_203].Status.eStatus= Burkert.eSensor_Status.HiHi_Alarm THEN tStatus:=eZ202_Status.PT203_High_Pressure_Alarm; END_IF;
//IF PVl.s8312[s8312_mapping.PT_203].Status.eStatus= Burkert.eSensor_Status.Low_Low_Alarm THEN tStatus:=eZ202_Status.PT203_Low_Pressure_Alarm; END_IF;

Test_Filters_P202_Level:=tStatus;




                
END_METHOD

METHOD Test_Filters_P203_Level : eZ202_Status
  VAR_INPUT
    Status : eZ202_status;
  END_VAR
  VAR
    tStatus : eZ202_Status;
  END_VAR
                  tStatus:=Status;
IF NOT(GVL.Filter_Path_Available) THEN tStatus:=eZ202_Status.No_Filter_Available; END_IF;


//IF NOT(GVL.s3363[s3363_mapping.ACV_203].Ready) 	THEN 	tStatus:=eZ202_Status.ACV203_Not_Ready; 	END_IF;
IF NOT(GVL.s3363[s3363_mapping.ACV_206].Ready) 	THEN 	tStatus:=eZ202_Status.ACV206_Not_Ready; 	END_IF;
//IF NOT(GVL.s3363[s3363_mapping.ACV_224].Ready) 	THEN 	tStatus:=eZ202_Status.ACV224_Not_Ready; 	END_IF;
//IF NOT(GVL.s3363[s3363_mapping.ACV_225].Ready) 	THEN 	tStatus:=eZ202_Status.ACV225_Not_Ready; 	END_IF;
IF NOT(GVL.s3363[s3363_mapping.ACV_226].Ready) 	THEN 	tStatus:=eZ202_Status.ACV226_Not_Ready; 	END_IF;

//IF NOT(Network.VFD[VFD_Mapping.VFD_202].Ready) 	THEN	tStatus:=eZ202_status.P202_Not_Ready;		END_IF;
IF NOT(Network.VFD[VFD_Mapping.VFD_203].Ready) 	THEN	tStatus:=eZ202_status.P203_Not_Ready;		END_IF;

IF NOT(PVL.Ait[AIT_Mapping.LT_202].Ready) 		THEN	tStatus:=eZ202_Status.LT202_Not_Ready;		END_IF;
//IF NOT(PVL.Ait[AIT_Mapping.LT_202A].Ready) 		THEN	tStatus:=eZ202_Status.LT202A_Not_Ready;		END_IF;

//IF NOT(PVl.s8312[s8312_mapping.PT_202].Ready)	THEN	tStatus:=ez202_Status.PT202_Not_Ready;		END_IF;
IF NOT(PVl.s8312[s8312_mapping.PT_203].Ready)	THEN	tStatus:=ez202_Status.PT203_Not_Ready;		END_IF;

IF NOT(PVL.s8098[s8098_mapping.FT_202].Ready)	THEN	tStatus:=ez202_Status.FT202_Not_Ready;		END_IF;
//IF NOT(PVL.s8098[s8098_mapping.FT_203].Ready)	THEN	tStatus:=ez202_Status.FT203_Not_Ready;		END_IF;
	
//IF gvl.LS[ls_mapping.LSLL_205].Status.eStatus=Burkert.DI_Status.No_Liquid_Detected_Alarm	THEN	tStatus:=eZ202_Status.P202_Intake_Empty;		END_IF;
IF gvl.LS[ls_mapping.LSLL_203].Status.eStatus=Burkert.DI_Status.No_Liquid_Detected_Alarm	THEN	tStatus:=eZ202_Status.P203_Intake_Empty;		END_IF;
//IF gvl.LS[ls_mapping.LSHH_201].Status.eStatus=Burkert.DI_Status.Liquid_Detected_Alarm		THEN	tStatus:=eZ202_Status.EP101_High_High_Alarm;	END_IF;




//IF GVL.s3363[s3363_mapping.ACV_203].Status.eStatus=Burkert.eACV_Status.Pos_Error THEN	tStatus:=eZ202_Status.ACV203_Error; END_IF;
IF GVL.s3363[s3363_mapping.ACV_206].Status.eStatus=Burkert.eACV_Status.Pos_Error THEN	tStatus:=eZ202_Status.ACV206_Error; END_IF;
//IF GVL.s3363[s3363_mapping.ACV_224].Status.eStatus=Burkert.eACV_Status.Pos_Error THEN	tStatus:=eZ202_Status.ACV224_Error; END_IF;
//IF GVL.s3363[s3363_mapping.ACV_225].Status.eStatus=Burkert.eACV_Status.Pos_Error THEN	tStatus:=eZ202_Status.ACV225_Error; END_IF;
IF GVL.s3363[s3363_mapping.ACV_226].Status.eStatus=Burkert.eACV_Status.Pos_Error THEN	tStatus:=eZ202_Status.ACV226_Error; END_IF;



IF PVL.AIT[AIT_Mapping.LT_202].Status.eStatus=Burkert.eSensor_Status.Low_Low_Alarm THEN	tStatus:=eZ202_Status.LT202_Low_Low_Alarm;	END_IF;

//IF PVL.AIT[AIT_Mapping.LT_202A].Status.eStatus=Burkert.eSensor_Status.Low_Low_Alarm THEN	tStatus:=eZ202_Status.LT202A_Low_Low_Alarm;	END_IF;

//IF (PVL.s8098[s8098_mapping.FT_202].PDO.VolumeFlow.Status.eStatus=burkert.eSensor_Status.Low_Low_Alarm)	THEN	tStatus:=ez202_Status.FT202_Low_Low_Flow_Alarm;		END_IF;
//IF (PVL.s8098[s8098_mapping.FT_202].PDO.VolumeFlow.Status.eStatus=burkert.eSensor_Status.HiHi_Alarm)	THEN	tStatus:=ez202_Status.FT202_High_High_Flow_Alarm;		END_IF;
//IF NOT(PVL.s8098[s8098_mapping.FT_203].PDO.VolumeFlow.Status.eStatus=burkert.eSensor_Status.Low_Low_Alarm)	THEN	tStatus:=ez202_Status.FT203_Low_Low_Flow_Alarm;		END_IF;
//IF NOT(PVL.s8098[s8098_mapping.FT_203].PDO.VolumeFlow.Status.eStatus=burkert.eSensor_Status.HiHi_Alarm)	THEN	tStatus:=ez202_Status.FT202_High_High_Flow_Alarm;		END_IF;
//IF (PVL.s8098[s8098_mapping.FT_202].PDO.VolumeFlow.Status.eStatus=burkert.eSensor_Status.Low_Low_Alarm)	THEN	tStatus:=ez202_Status.FT202_Low_Low_Flow_Alarm;		END_IF;
//IF (PVL.s8098[s8098_mapping.FT_202].PDO.VolumeFlow.Status.eStatus=burkert.eSensor_Status.HiHi_Alarm)	THEN	tStatus:=ez202_Status.FT202_High_High_Flow_Alarm;		END_IF;
//IF (PVL.s8098[s8098_mapping.FT_203].PDO.VolumeFlow.Status.eStatus=burkert.eSensor_Status.Low_Low_Alarm)	THEN	tStatus:=ez202_Status.FT203_Low_Low_Flow_Alarm;		END_IF;
//IF (PVL.s8098[s8098_mapping.FT_203].PDO.VolumeFlow.Status.eStatus=burkert.eSensor_Status.HiHi_Alarm)	THEN	tStatus:=ez202_Status.FT202_High_High_Flow_Alarm;		END_IF;


IF PVl.s8312[s8312_mapping.PT_202].Status.eStatus= Burkert.eSensor_Status.HiHi_Alarm THEN tStatus:=eZ202_Status.PT202_High_Pressure_Alarm; END_IF;
IF PVl.s8312[s8312_mapping.PT_202].Status.eStatus= Burkert.eSensor_Status.Low_Low_Alarm THEN tStatus:=eZ202_Status.PT202_Low_Pressure_Alarm; END_IF;
//IF PVl.s8312[s8312_mapping.PT_203].Status.eStatus= Burkert.eSensor_Status.HiHi_Alarm THEN tStatus:=eZ202_Status.PT203_High_Pressure_Alarm; END_IF;
//IF PVl.s8312[s8312_mapping.PT_203].Status.eStatus= Burkert.eSensor_Status.Low_Low_Alarm THEN tStatus:=eZ202_Status.PT203_Low_Pressure_Alarm; END_IF;

Test_Filters_P203_Level:=tStatus;




                
END_METHOD

METHOD Test_Z201_Return_P202_Level : eZ202_Status
  VAR_INPUT
    Status : eZ202_status;
  END_VAR
  VAR
    tStatus : eZ202_Status;
  END_VAR
                  tStatus:=Status;


IF NOT(GVL.s3363[s3363_mapping.ACV_203].Ready) 	THEN 	tStatus:=eZ202_Status.ACV203_Not_Ready; 	END_IF;
IF NOT(GVL.s3363[s3363_mapping.ACV_206].Ready) 	THEN 	tStatus:=eZ202_Status.ACV206_Not_Ready; 	END_IF;
//IF NOT(GVL.s3363[s3363_mapping.ACV_224].Ready) 	THEN 	tStatus:=eZ202_Status.ACV224_Not_Ready; 	END_IF;
//IF NOT(GVL.s3363[s3363_mapping.ACV_225].Ready) 	THEN 	tStatus:=eZ202_Status.ACV225_Not_Ready; 	END_IF;
IF NOT(GVL.s3363[s3363_mapping.ACV_226].Ready) 	THEN 	tStatus:=eZ202_Status.ACV226_Not_Ready; 	END_IF;

IF NOT(Network.VFD[VFD_Mapping.VFD_202].Ready) 	THEN	tStatus:=eZ202_status.P202_Not_Ready;		END_IF;
//IF NOT(Network.VFD[VFD_Mapping.VFD_203].Ready) 	THEN	tStatus:=eZ202_status.P203_Not_Ready;		END_IF;

IF NOT(PVL.Ait[AIT_Mapping.LT_202].Ready) 		THEN	tStatus:=eZ202_Status.LT202_Not_Ready;		END_IF;
//IF NOT(PVL.Ait[AIT_Mapping.LT_202A].Ready) 		THEN	tStatus:=eZ202_Status.LT202A_Not_Ready;		END_IF;

///////********		IF NOT(PVl.s8312[s8312_mapping.PT_202].Ready)	THEN	tStatus:=ez202_Status.PT202_Not_Ready;		END_IF;
///////********		IF NOT(PVl.s8312[s8312_mapping.PT_203].Ready)	THEN	tStatus:=ez202_Status.PT203_Not_Ready;		END_IF;

//IF NOT(PVL.s8098[s8098_mapping.FT_202].Ready)	THEN	tStatus:=ez202_Status.FT202_Not_Ready;		END_IF;
//IF NOT(PVL.s8098[s8098_mapping.FT_203].Ready)	THEN	tStatus:=ez202_Status.FT203_Not_Ready;		END_IF;
	
IF gvl.LS[ls_mapping.LSLL_205].Status.eStatus=Burkert.DI_Status.No_Liquid_Detected_Alarm	THEN	tStatus:=eZ202_Status.P202_Intake_Empty;		END_IF;
//IF gvl.LS[ls_mapping.LSLL_203].Status.eStatus=Burkert.DI_Status.No_Liquid_Detected_Alarm	THEN	tStatus:=eZ202_Status.P203_Intake_Empty;		END_IF;
IF gvl.LS[ls_mapping.LSHH_201].Status.eStatus=Burkert.DI_Status.Liquid_Detected_Alarm		THEN	tStatus:=eZ202_Status.EP101_High_High_Alarm;	END_IF;

//IF NOT(PVL.Ait[AIT_Mapping.LT_202].Ready) 		THEN	tStatus:=eZ202_Status.LT202_Not_Ready;		END_IF;
//IF (PVL.Ait[AIT_Mapping.LT_202].Status.eStatus=Burkert.eSensor_Status.HiHi_Alarm) 		THEN	tStatus:=eZ202_Status.LT202_High_High_Alarm;		END_IF;

IF NOT(PVL.Ait[AIT_Mapping.LT_201].Ready) 		THEN	tStatus:=eZ202_Status.LT201_Not_Ready;		END_IF;
IF (PVL.Ait[AIT_Mapping.LT_201].Status.eStatus=Burkert.eSensor_Status.HiHi_Alarm) 		THEN	tStatus:=eZ202_Status.LT201_High_High_Alarm;		END_IF;

IF NOT(pVL.Ait[AIT_Mapping.LT_101_P].Ready) 		THEN	tStatus:=eZ202_Status.LT101_Not_Ready;		END_IF;
IF (PVL.Ait[AIT_Mapping.LT_101_P].Status.eStatus=Burkert.eSensor_Status.HiHi_Alarm) 		THEN	tStatus:=eZ202_Status.LT101_High_High_Alarm;		END_IF;

//IF (PVL.Ait[AIT_Mapping.LT_202A].Ready) 		THEN	tStatus:=eZ202_Status.LT202A_Not_Ready;		END_IF;


IF GVL.s3363[s3363_mapping.ACV_203].Status.eStatus=Burkert.eACV_Status.Pos_Error THEN	tStatus:=eZ202_Status.ACV203_Error; END_IF;
IF GVL.s3363[s3363_mapping.ACV_206].Status.eStatus=Burkert.eACV_Status.Pos_Error THEN	tStatus:=eZ202_Status.ACV206_Error; END_IF;
//IF GVL.s3363[s3363_mapping.ACV_224].Status.eStatus=Burkert.eACV_Status.Pos_Error THEN	tStatus:=eZ202_Status.ACV224_Error; END_IF;
//IF GVL.s3363[s3363_mapping.ACV_225].Status.eStatus=Burkert.eACV_Status.Pos_Error THEN	tStatus:=eZ202_Status.ACV225_Error; END_IF;
IF GVL.s3363[s3363_mapping.ACV_226].Status.eStatus=Burkert.eACV_Status.Pos_Error THEN	tStatus:=eZ202_Status.ACV226_Error; END_IF;

//IF NOT(GVL.Filter_Path_Available) THEN tStatus:=eZ202_Status.No_Filter_Available; END_IF;

//IF (PVL.s8098[s8098_mapping.FT_202].PDO.VolumeFlow.Status.eStatus=burkert.eSensor_Status.Low_Low_Alarm)	THEN	tStatus:=ez202_Status.FT202_Low_Low_Flow_Alarm;		END_IF;
//IF (PVL.s8098[s8098_mapping.FT_202].PDO.VolumeFlow.Status.eStatus=burkert.eSensor_Status.HiHi_Alarm)	THEN	tStatus:=ez202_Status.FT202_High_High_Flow_Alarm;		END_IF;
//IF (PVL.s8098[s8098_mapping.FT_203].PDO.VolumeFlow.Status.eStatus=burkert.eSensor_Status.Low_Low_Alarm)	THEN	tStatus:=ez202_Status.FT203_Low_Low_Flow_Alarm;		END_IF;
//IF (PVL.s8098[s8098_mapping.FT_203].PDO.VolumeFlow.Status.eStatus=burkert.eSensor_Status.HiHi_Alarm)	THEN	tStatus:=ez202_Status.FT202_High_High_Flow_Alarm;		END_IF;


//IF PVl.s8312[s8312_mapping.PT_202].Status.eStatus= Burkert.eSensor_Status.HiHi_Alarm THEN tStatus:=eZ202_Status.PT202_High_Pressure_Alarm; END_IF;
//IF PVl.s8312[s8312_mapping.PT_202].Status.eStatus= Burkert.eSensor_Status.Low_Low_Alarm THEN tStatus:=eZ202_Status.PT202_Low_Pressure_Alarm; END_IF;
///////********		IF PVl.s8312[s8312_mapping.PT_203].Status.eStatus= Burkert.eSensor_Status.HiHi_Alarm THEN tStatus:=eZ202_Status.PT203_High_Pressure_Alarm; END_IF;
///////********		IF PVl.s8312[s8312_mapping.PT_203].Status.eStatus= Burkert.eSensor_Status.Low_Low_Alarm THEN tStatus:=eZ202_Status.PT203_Low_Pressure_Alarm; END_IF;

IF (PVL.Ait[AIT_Mapping.LT_202].Status.eStatus=Burkert.eSensor_Status.Low_Low_Alarm) 		THEN	tStatus:=eZ202_Status.LT202_Low_Low_Alarm;		END_IF;

Test_Z201_Return_P202_Level:=tStatus;
                
END_METHOD

METHOD Test_Z201_Return_P203_Level : eZ202_Status
  VAR_INPUT
    Status : eZ202_status;
  END_VAR
  VAR
    tStatus : eZ202_Status;
  END_VAR
                  tStatus:=Status;


IF NOT(GVL.s3363[s3363_mapping.ACV_203].Ready) 	THEN 	tStatus:=eZ202_Status.ACV203_Not_Ready; 	END_IF;
//IF NOT(GVL.s3363[s3363_mapping.ACV_206].Ready) 	THEN 	tStatus:=eZ202_Status.ACV206_Not_Ready; 	END_IF;
//IF NOT(GVL.s3363[s3363_mapping.ACV_224].Ready) 	THEN 	tStatus:=eZ202_Status.ACV224_Not_Ready; 	END_IF;
//IF NOT(GVL.s3363[s3363_mapping.ACV_225].Ready) 	THEN 	tStatus:=eZ202_Status.ACV225_Not_Ready; 	END_IF;
IF NOT(GVL.s3363[s3363_mapping.ACV_226].Ready) 	THEN 	tStatus:=eZ202_Status.ACV226_Not_Ready; 	END_IF;

//IF NOT(Network.VFD[VFD_Mapping.VFD_202].Ready) 	THEN	tStatus:=eZ202_status.P202_Not_Ready;		END_IF;
IF NOT(Network.VFD[VFD_Mapping.VFD_203].Ready) 	THEN	tStatus:=eZ202_status.P203_Not_Ready;		END_IF;

IF NOT(PVL.Ait[AIT_Mapping.LT_202].Ready) 		THEN	tStatus:=eZ202_Status.LT202_Not_Ready;		END_IF;
//IF NOT(PVL.Ait[AIT_Mapping.LT_202A].Ready) 		THEN	tStatus:=eZ202_Status.LT202A_Not_Ready;		END_IF;

//IF NOT(PVl.s8312[s8312_mapping.PT_202].Ready)	THEN	tStatus:=ez202_Status.PT202_Not_Ready;		END_IF;
///////********		IF NOT(PVl.s8312[s8312_mapping.PT_203].Ready)	THEN	tStatus:=ez202_Status.PT203_Not_Ready;		END_IF;

//IF NOT(PVL.s8098[s8098_mapping.FT_202].Ready)	THEN	tStatus:=ez202_Status.FT202_Not_Ready;		END_IF;
//IF NOT(PVL.s8098[s8098_mapping.FT_203].Ready)	THEN	tStatus:=ez202_Status.FT203_Not_Ready;		END_IF;
	
//IF gvl.LS[ls_mapping.LSLL_205].Status.eStatus=Burkert.DI_Status.No_Liquid_Detected_Alarm	THEN	tStatus:=eZ202_Status.P202_Intake_Empty;		END_IF;
IF gvl.LS[ls_mapping.LSLL_203].Status.eStatus=Burkert.DI_Status.No_Liquid_Detected_Alarm	THEN	tStatus:=eZ202_Status.P203_Intake_Empty;		END_IF;
IF gvl.LS[ls_mapping.LSHH_201].Status.eStatus=Burkert.DI_Status.Liquid_Detected_Alarm		THEN	tStatus:=eZ202_Status.EP101_High_High_Alarm;	END_IF;

//IF NOT(PVL.Ait[AIT_Mapping.LT_202].Ready) 		THEN	tStatus:=eZ202_Status.LT202_Not_Ready;		END_IF;
//IF (PVL.Ait[AIT_Mapping.LT_202].Status.eStatus=Burkert.eSensor_Status.HiHi_Alarm) 		THEN	tStatus:=eZ202_Status.LT202_High_High_Alarm;		END_IF;

IF NOT(PVL.Ait[AIT_Mapping.LT_201].Ready) 		THEN	tStatus:=eZ202_Status.LT201_Not_Ready;		END_IF;
IF (PVL.Ait[AIT_Mapping.LT_201].Status.eStatus=Burkert.eSensor_Status.HiHi_Alarm) 		THEN	tStatus:=eZ202_Status.LT201_High_High_Alarm;		END_IF;

IF NOT(PVL.Ait[AIT_Mapping.LT_101_p].Ready) 		THEN	tStatus:=eZ202_Status.LT101_Not_Ready;		END_IF;
IF (PVL.Ait[AIT_Mapping.LT_101_P].Status.eStatus=Burkert.eSensor_Status.HiHi_Alarm) 		THEN	tStatus:=eZ202_Status.LT101_High_High_Alarm;		END_IF;


IF GVL.s3363[s3363_mapping.ACV_203].Status.eStatus=Burkert.eACV_Status.Pos_Error THEN	tStatus:=eZ202_Status.ACV203_Error; END_IF;
//IF GVL.s3363[s3363_mapping.ACV_206].Status.eStatus=Burkert.eACV_Status.Pos_Error THEN	tStatus:=eZ202_Status.ACV206_Error; END_IF;
//IF GVL.s3363[s3363_mapping.ACV_224].Status.eStatus=Burkert.eACV_Status.Pos_Error THEN	tStatus:=eZ202_Status.ACV224_Error; END_IF;
//IF GVL.s3363[s3363_mapping.ACV_225].Status.eStatus=Burkert.eACV_Status.Pos_Error THEN	tStatus:=eZ202_Status.ACV225_Error; END_IF;
IF GVL.s3363[s3363_mapping.ACV_226].Status.eStatus=Burkert.eACV_Status.Pos_Error THEN	tStatus:=eZ202_Status.ACV226_Error; END_IF;

//IF NOT(GVL.Filter_Path_Available) THEN tStatus:=eZ202_Status.No_Filter_Available; END_IF;

//IF (PVL.s8098[s8098_mapping.FT_202].PDO.VolumeFlow.Status.eStatus=burkert.eSensor_Status.Low_Low_Alarm)	THEN	tStatus:=ez202_Status.FT202_Low_Low_Flow_Alarm;		END_IF;
//IF (PVL.s8098[s8098_mapping.FT_202].PDO.VolumeFlow.Status.eStatus=burkert.eSensor_Status.HiHi_Alarm)	THEN	tStatus:=ez202_Status.FT202_High_High_Flow_Alarm;		END_IF;
//IF (PVL.s8098[s8098_mapping.FT_203].PDO.VolumeFlow.Status.eStatus=burkert.eSensor_Status.Low_Low_Alarm)	THEN	tStatus:=ez202_Status.FT203_Low_Low_Flow_Alarm;		END_IF;
//IF (PVL.s8098[s8098_mapping.FT_203].PDO.VolumeFlow.Status.eStatus=burkert.eSensor_Status.HiHi_Alarm)	THEN	tStatus:=ez202_Status.FT202_High_High_Flow_Alarm;		END_IF;


//IF PVl.s8312[s8312_mapping.PT_202].Status.eStatus= Burkert.eSensor_Status.HiHi_Alarm THEN tStatus:=eZ202_Status.PT202_High_Pressure_Alarm; END_IF;
//IF PVl.s8312[s8312_mapping.PT_202].Status.eStatus= Burkert.eSensor_Status.Low_Low_Alarm THEN tStatus:=eZ202_Status.PT202_Low_Pressure_Alarm; END_IF;
///////********		IF PVl.s8312[s8312_mapping.PT_203].Status.eStatus= Burkert.eSensor_Status.HiHi_Alarm THEN tStatus:=eZ202_Status.PT203_High_Pressure_Alarm; END_IF;
///////********		IF PVl.s8312[s8312_mapping.PT_203].Status.eStatus= Burkert.eSensor_Status.Low_Low_Alarm THEN tStatus:=eZ202_Status.PT203_Low_Pressure_Alarm; END_IF;


IF (PVL.Ait[AIT_Mapping.LT_202].Status.eStatus=Burkert.eSensor_Status.Low_Low_Alarm) 		THEN	tStatus:=eZ202_Status.LT202_Low_Low_Alarm;		END_IF;
Test_Z201_Return_p203_Level:=tStatus;
                
END_METHOD
END_PROGRAM

PROGRAM CanOpen_IO
  VAR
    ME64_001_CTRL : Burkert.CanOpen_ME64;
    BCV_001_CTRL : Burkert.CanOpen_8691;
    ACV_001_CTRL : Burkert.CanOpen_8694;
    b8653_001_CTRL : Burkert.CanOpen_8653;
  END_VAR

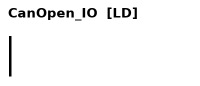
(* LD diagram, written out as Structured Text *)
END_PROGRAM

PROGRAM DI_Manager
  VAR
    External_Pump_Status : Burkert.DI_UDFB;
    DC_OK : Burkert.DI_UDFB;
    Z201_DC_OK : Burkert.DI_UDFB;
  END_VAR

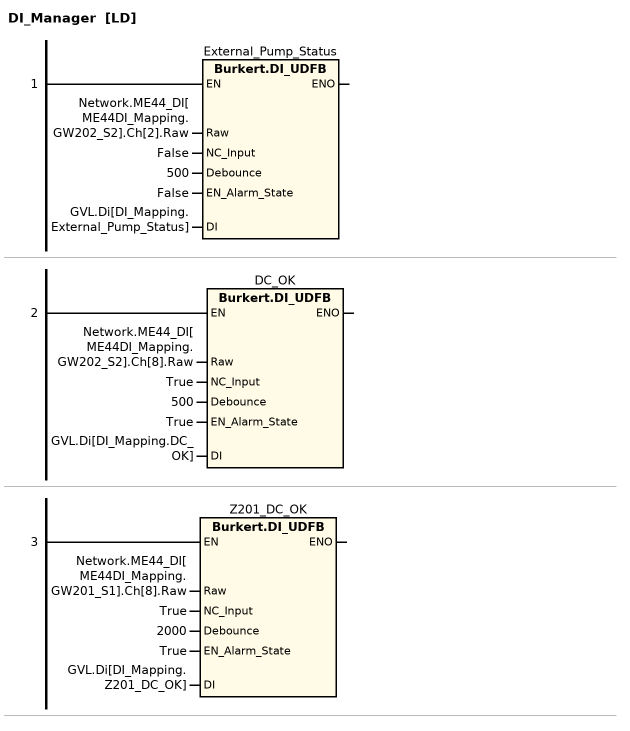
(* LD diagram, written out as Structured Text *)

External_Pump_Status(Raw := Network.ME44_DI[ME44DI_Mapping.GW202_S2].Ch[2].Raw, NC_Input := False, Debounce := 500, EN_Alarm_State := False, DI := GVL.Di[DI_Mapping.External_Pump_Status]);

DC_OK(Raw := Network.ME44_DI[ME44DI_Mapping.GW202_S2].Ch[8].Raw, NC_Input := True, Debounce := 500, EN_Alarm_State := True, DI := GVL.Di[DI_Mapping.DC_OK]);

Z201_DC_OK(Raw := Network.ME44_DI[ME44DI_Mapping.GW201_S1].Ch[8].Raw, NC_Input := True, Debounce := 2000, EN_Alarm_State := True, DI := GVL.Di[DI_Mapping.Z201_DC_OK]);
END_PROGRAM

PROGRAM PT_Manager
  VAR
    PT101_CTRL : Burkert.eDip_8312;
    PT201_CTRL : Burkert.eDip_8312;
    PT202_CTRL : Burkert.eDip_8312;
    PT203_CTRL : Burkert.eDip_8312;
    PT204_CTRL : Burkert.eDip_8312;
    PT205_CTRL : Burkert.eDip_8312;
  END_VAR

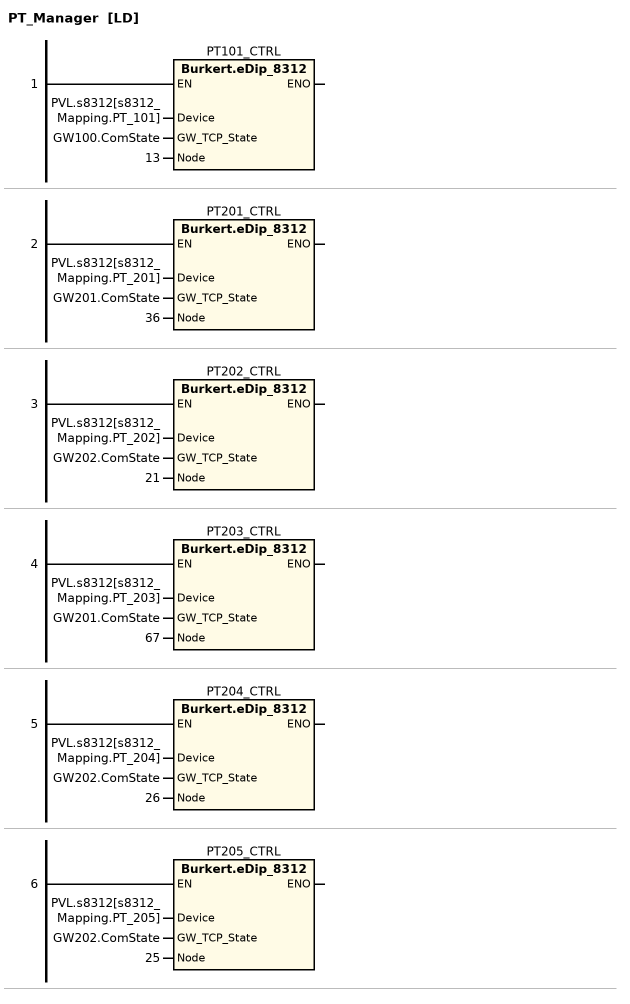
(* LD diagram, written out as Structured Text *)

PT101_CTRL(Device := PVL.s8312[s8312_Mapping.PT_101], GW_TCP_State := GW100.ComState, Node := 13);

PT201_CTRL(Device := PVL.s8312[s8312_Mapping.PT_201], GW_TCP_State := GW201.ComState, Node := 36);

PT202_CTRL(Device := PVL.s8312[s8312_Mapping.PT_202], GW_TCP_State := GW202.ComState, Node := 21);

PT203_CTRL(Device := PVL.s8312[s8312_Mapping.PT_203], GW_TCP_State := GW201.ComState, Node := 67);

PT204_CTRL(Device := PVL.s8312[s8312_Mapping.PT_204], GW_TCP_State := GW202.ComState, Node := 26);

PT205_CTRL(Device := PVL.s8312[s8312_Mapping.PT_205], GW_TCP_State := GW202.ComState, Node := 25);
END_PROGRAM

PROGRAM MEx3_ORF
  VAR
    GW_Z100 : Burkert.ME43_SDO;
    GW_Z201 : Burkert.ME43_SDO;
    GW_Z202 : Burkert.ME43_SDO;
    GW_TK201 : Burkert.ME43_SDO;
  END_VAR

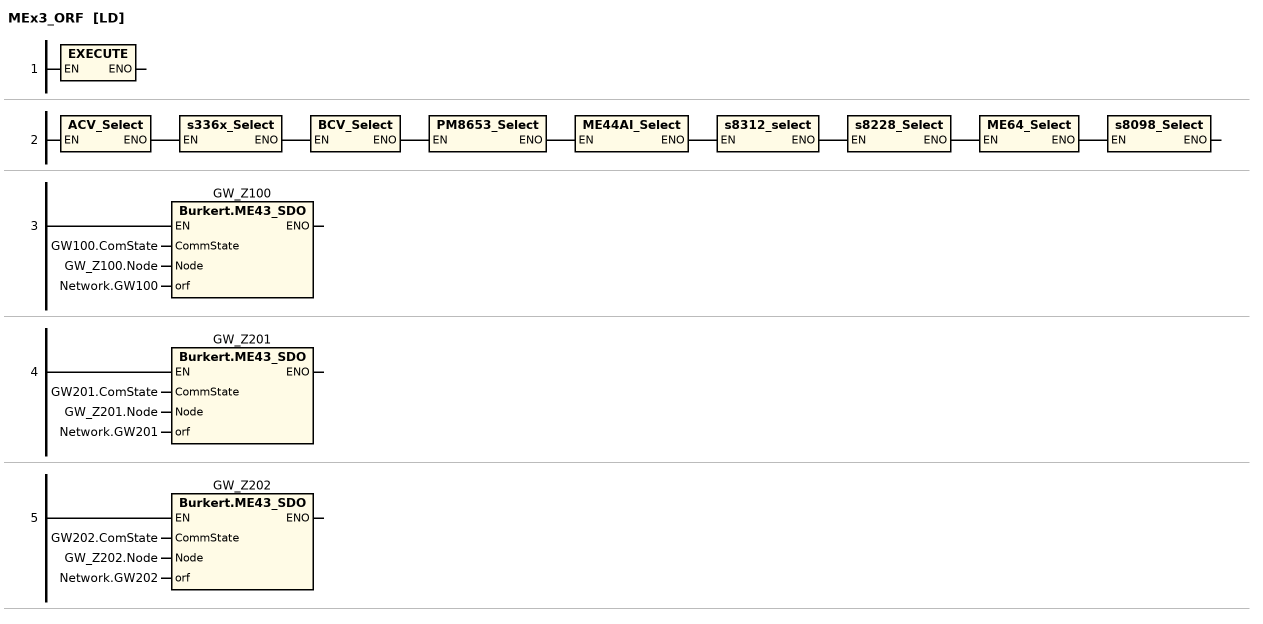
(* LD diagram, written out as Structured Text *)

GW_Z100.Node:=255;
GW_Z201.Node:=255;
GW_Z202.Node:=255;
GW_TK201.Node:=255;

ACV_Select();
s336x_Select();
BCV_Select();
PM8653_Select();
ME44AI_Select();
s8312_select();
s8228_Select();
ME64_Select();
s8098_Select();

GW_Z100(CommState := GW100.ComState, Node := GW_Z100.Node, orf := Network.GW100);

GW_Z201(CommState := GW201.ComState, Node := GW_Z201.Node, orf := Network.GW201);

GW_Z202(CommState := GW202.ComState, Node := GW_Z202.Node, orf := Network.GW202);

ACTION s8098_Select:
                CASE HMI.HMI_8098_Index OF
	
	s8098_Mapping.FT_101:	GW_Z100.r8098 REF= 	pvl.s8098[HMI.HMI_8098_Index];
							GW_Z100.Node:=	pvl.s8098[HMI.HMI_8098_Index].DSO.Node;
							
	s8098_Mapping.FT_201:	GW_Z201.r8098 REF= 	pvl.s8098[HMI.HMI_8098_Index];
							GW_Z201.Node:=	pvl.s8098[HMI.HMI_8098_Index].DSO.Node;
	
	s8098_Mapping.FT_202:	GW_Z202.r8098 REF= 	pvl.s8098[HMI.HMI_8098_Index];
							GW_Z202.Node:=	pvl.s8098[HMI.HMI_8098_Index].DSO.Node;
							
	s8098_Mapping.FT_203:	GW_Z201.r8098 REF= 	pvl.s8098[HMI.HMI_8098_Index];
							GW_Z201.Node:=	pvl.s8098[HMI.HMI_8098_Index].DSO.Node;
							
	s8098_Mapping.FT_204:	GW_Z202.r8098 REF= 	pvl.s8098[HMI.HMI_8098_Index];
							GW_Z202.Node:=	pvl.s8098[HMI.HMI_8098_Index].DSO.Node;

END_CASE
              
END_ACTION

ACTION ME64_Select:
                CASE HMI.ME64_Index OF
	(*
	ME64_mapping.Branch_1:	GW_Branch_1.Node:=Network.Branch_1_ME64.DSO.Node; GW_Branch_1.rME64 REF= Network.Branch_1_ME64; Burkert.HMI_ME64_Sync(Local:=Network.Branch_1_ME64,HMI:=HMI.ME64_Data);
	ME64_mapping.Branch_2:	GW_Branch_2.Node:=Network.Branch_2_ME64.DSO.Node; GW_Branch_2.rME64 REF= Network.Branch_2_ME64;	Burkert.HMI_ME64_Sync(Local:=Network.Branch_2_ME64,HMI:=HMI.ME64_Data);
	ME64_mapping.Branch_3:	GW_Branch_3.Node:=Network.Branch_3_ME64.DSO.Node; GW_Branch_3.rME64 REF= Network.Branch_3_ME64;	Burkert.HMI_ME64_Sync(Local:=Network.Branch_3_ME64,HMI:=HMI.ME64_Data);
	ME64_mapping.Branch_4:	GW_Branch_4.Node:=Network.Branch_4_ME64.DSO.Node; GW_Branch_4.rME64 REF= Network.Branch_4_ME64;	Burkert.HMI_ME64_Sync(Local:=Network.Branch_4_ME64,HMI:=HMI.ME64_Data);
	ME64_mapping.Branch_5:	GW_Branch_5.Node:=Network.Branch_5_ME64.DSO.Node; GW_Branch_5.rME64 REF= Network.Branch_5_ME64;	Burkert.HMI_ME64_Sync(Local:=Network.Branch_5_ME64,HMI:=HMI.ME64_Data);
	ME64_mapping.Branch_6:	GW_Branch_6.Node:=Network.Branch_6_ME64.DSO.Node; GW_Branch_6.rME64 REF= Network.Branch_6_ME64;	Burkert.HMI_ME64_Sync(Local:=Network.Branch_6_ME64,HMI:=HMI.ME64_Data);
	
	ME64_mapping.CWS:	GW_CWS.Node:=Network.CWS_ME64.DSO.Node; 	GW_CWS.rME64 REF= Network.CWS_ME64;			Burkert.HMI_ME64_Sync(Local:=Network.CWS_ME64,HMI:=HMI.ME64_Data);
	ME64_mapping.HWS:	GW_HWS.Node:=Network.HWS_ME64.DSO.Node; 	GW_HWS.rME64 REF= Network.HWS_ME64;			Burkert.HMI_ME64_Sync(Local:=Network.HWS_ME64,HMI:=HMI.ME64_Data);
	ME64_mapping.RO:	GW_RO.Node:=Network.RO_ME64_10 .DSO.Node; 	GW_RO.rME64 REF= Network.RO_ME64_10;		Burkert.HMI_ME64_Sync(Local:=Network.RO_ME64_10,HMI:=HMI.ME64_Data);
	ME64_mapping.Brine:	GW_Brine.Node:=Network.Brine_ME64.DSO.Node; GW_Brine.rME64 REF= Network.Brine_ME64;	Burkert.HMI_ME64_Sync(Local:=Network.Brine_ME64,HMI:=HMI.ME64_Data);
	*)
END_CASE
              
END_ACTION

ACTION BCV_Select:
                CASE HMI.HMI_BCV_Index OF
	(*
	BCV_Mapping.Branch_1_Brine_Pump_Discharge:	GW_Branch_1.r8691 REF= GVL.BCV[BCV_Mapping.Branch_1_Brine_Pump_Discharge]; 	Gw_branch_1.Node:=GVL.BCV[BCV_Mapping.Branch_1_Brine_Pump_Discharge].DSO.Node; 
	BCV_Mapping.Branch_1_Brine_Pump_Flush:		GW_Branch_1.r8691 REF= GVL.BCV[BCV_Mapping.Branch_1_Brine_Pump_Flush]; 		Gw_branch_1.Node:=GVL.BCV[BCV_Mapping.Branch_1_Brine_Pump_Flush].DSO.Node; 
	BCV_Mapping.Branch_1_Brine_Pump_Supply:		GW_Branch_1.r8691 REF= GVL.BCV[BCV_Mapping.Branch_1_Brine_Pump_Supply]; 	Gw_branch_1.Node:=GVL.BCV[BCV_Mapping.Branch_1_Brine_Pump_Supply].DSO.Node;
	
	BCV_Mapping.Branch_2_Brine_Pump_Discharge:	GW_Branch_2.r8691 REF= GVL.BCV[BCV_Mapping.Branch_2_Brine_Pump_Discharge]; 	Gw_branch_2.Node:=GVL.BCV[BCV_Mapping.Branch_2_Brine_Pump_Discharge].DSO.Node; 
	BCV_Mapping.Branch_2_Brine_Pump_Flush:		GW_Branch_2.r8691 REF= GVL.BCV[BCV_Mapping.Branch_2_Brine_Pump_Flush]; 		Gw_branch_2.Node:=GVL.BCV[BCV_Mapping.Branch_2_Brine_Pump_Flush].DSO.Node; 
	BCV_Mapping.Branch_2_Brine_Pump_Supply:		GW_Branch_2.r8691 REF= GVL.BCV[BCV_Mapping.Branch_2_Brine_Pump_Supply]; 	Gw_branch_2.Node:=GVL.BCV[BCV_Mapping.Branch_2_Brine_Pump_Supply].DSO.Node; 
	
	BCV_Mapping.Branch_3_Brine_Pump_Discharge:	GW_Branch_3.r8691 REF= GVL.BCV[BCV_Mapping.Branch_3_Brine_Pump_Discharge]; 	Gw_branch_3.Node:=GVL.BCV[BCV_Mapping.Branch_3_Brine_Pump_Discharge].DSO.Node; 
	BCV_Mapping.Branch_3_Brine_Pump_Flush:		GW_Branch_3.r8691 REF= GVL.BCV[BCV_Mapping.Branch_3_Brine_Pump_Flush]; 		Gw_branch_3.Node:=GVL.BCV[BCV_Mapping.Branch_3_Brine_Pump_Flush].DSO.Node; 
	BCV_Mapping.Branch_3_Brine_Pump_Supply:		GW_Branch_3.r8691 REF= GVL.BCV[BCV_Mapping.Branch_3_Brine_Pump_Supply]; 	Gw_branch_3.Node:=GVL.BCV[BCV_Mapping.Branch_3_Brine_Pump_Supply].DSO.Node; 
	
	BCV_Mapping.Branch_4_Brine_Pump_Discharge:	GW_Branch_4.r8691 REF= GVL.BCV[BCV_Mapping.Branch_4_Brine_Pump_Discharge]; 	Gw_branch_4.Node:=GVL.BCV[BCV_Mapping.Branch_4_Brine_Pump_Discharge].DSO.Node; 
	BCV_Mapping.Branch_4_Brine_Pump_Flush:		GW_Branch_4.r8691 REF= GVL.BCV[BCV_Mapping.Branch_4_Brine_Pump_Flush]; 		Gw_branch_4.Node:=GVL.BCV[BCV_Mapping.Branch_4_Brine_Pump_Flush].DSO.Node; 
	BCV_Mapping.Branch_4_Brine_Pump_Supply:		GW_Branch_4.r8691 REF= GVL.BCV[BCV_Mapping.Branch_4_Brine_Pump_Supply]; 	Gw_branch_4.Node:=GVL.BCV[BCV_Mapping.Branch_4_Brine_Pump_Supply].DSO.Node; 

	BCV_Mapping.Branch_5_Brine_Pump_Discharge:	GW_Branch_5.r8691 REF= GVL.BCV[BCV_Mapping.Branch_5_Brine_Pump_Discharge]; Gw_branch_5.Node:=GVL.BCV[BCV_Mapping.Branch_5_Brine_Pump_Discharge].DSO.Node; 
	BCV_Mapping.Branch_5_Brine_Pump_Flush:		GW_Branch_5.r8691 REF= GVL.BCV[BCV_Mapping.Branch_5_Brine_Pump_Flush]; Gw_branch_5.Node:=GVL.BCV[BCV_Mapping.Branch_5_Brine_Pump_Flush].DSO.Node; 
	BCV_Mapping.Branch_5_Brine_Pump_Supply:		GW_Branch_5.r8691 REF= GVL.BCV[BCV_Mapping.Branch_5_Brine_Pump_Supply]; Gw_branch_5.Node:=GVL.BCV[BCV_Mapping.Branch_5_Brine_Pump_Supply].DSO.Node; 
	
	BCV_Mapping.TK203_Bottom_Discharge_Valve :		GW_brine.r8691 REF= GVL.BCV[BCV_Mapping.TK203_Bottom_Discharge_Valve]; 				GW_brine.Node:=GVL.BCV[BCV_Mapping.TK203_Bottom_Discharge_Valve].DSO.Node; 
	BCV_Mapping.TK203_CIP_Chemical_Valve :			GW_brine.r8691 REF= GVL.BCV[BCV_Mapping.TK203_CIP_Chemical_Valve]; 					GW_brine.Node:=GVL.BCV[BCV_Mapping.TK203_CIP_Chemical_Valve].DSO.Node; 
	BCV_Mapping.TK203_LP_Drain_Valve :				GW_brine.r8691 REF= GVL.BCV[BCV_Mapping.TK203_LP_Drain_Valve]; 						GW_brine.Node:=GVL.BCV[BCV_Mapping.TK203_LP_Drain_Valve].DSO.Node; 
	BCV_Mapping.TK203_RO_Water_MakeUp_Flow_Valve :		GW_brine.r8691 REF= GVL.BCV[BCV_Mapping.TK203_RO_Water_MakeUp_Flow_Valve]; 		GW_brine.Node:=GVL.BCV[BCV_Mapping.TK203_RO_Water_MakeUp_Flow_Valve].DSO.Node; 
	BCV_Mapping.TK203_Side_Discharge_Valve :		GW_brine.r8691 REF= GVL.BCV[BCV_Mapping.TK203_Side_Discharge_Valve]; 				GW_brine.Node:=GVL.BCV[BCV_Mapping.TK203_Side_Discharge_Valve].DSO.Node; 
	
	*)
END_CASE
              
END_ACTION

ACTION s8228_Select:
                CASE HMI.HMI_8228_Index OF
	(*
	s8228_mapping.Branch_1:	GW_Branch_1.Node:=PVL.s8228[HMI.HMI_8228_Index].DSO.Node; GW_Branch_1.r8228 REF=PVL.s8228[HMI.HMI_8228_Index];
	s8228_mapping.Branch_2:	GW_Branch_2.Node:=PVL.s8228[HMI.HMI_8228_Index].DSO.Node; GW_Branch_2.r8228 REF=PVL.s8228[HMI.HMI_8228_Index];
	s8228_mapping.Branch_3:	GW_Branch_3.Node:=PVL.s8228[HMI.HMI_8228_Index].DSO.Node; GW_Branch_3.r8228 REF=PVL.s8228[HMI.HMI_8228_Index];
	s8228_mapping.Branch_4:	GW_Branch_4.Node:=PVL.s8228[HMI.HMI_8228_Index].DSO.Node; GW_Branch_4.r8228 REF=PVL.s8228[HMI.HMI_8228_Index];
	s8228_mapping.Branch_5:	GW_Branch_5.Node:=PVL.s8228[HMI.HMI_8228_Index].DSO.Node; GW_Branch_5.r8228 REF=PVL.s8228[HMI.HMI_8228_Index];
	s8228_mapping.Branch_6:	GW_Branch_6.Node:=PVL.s8228[HMI.HMI_8228_Index].DSO.Node; GW_Branch_6.r8228 REF=PVL.s8228[HMI.HMI_8228_Index];
	
	*)
END_CASE
              
END_ACTION

ACTION s8312_select:
                CASE HMI.HMI_8312_Index OF
	

	s8312_mapping.PT_101:	GW_Z100.Node:=PVl.s8312[HMI.HMI_8312_Index].DSO.Node; GW_Z100.r8312 REF=PVl.s8312[HMI.HMI_8312_Index];
	s8312_mapping.PT_201:	GW_Z201.Node:=PVl.s8312[HMI.HMI_8312_Index].DSO.Node; GW_Z201.r8312 REF=PVl.s8312[HMI.HMI_8312_Index];
	s8312_mapping.PT_202:	GW_Z202.Node:=PVl.s8312[HMI.HMI_8312_Index].DSO.Node; GW_Z202.r8312 REF=PVl.s8312[HMI.HMI_8312_Index];
	s8312_mapping.PT_204:	GW_Z202.Node:=PVl.s8312[HMI.HMI_8312_Index].DSO.Node; GW_Z202.r8312 REF=PVl.s8312[HMI.HMI_8312_Index];
	s8312_mapping.PT_205:	GW_Z202.Node:=PVl.s8312[HMI.HMI_8312_Index].DSO.Node; GW_Z202.r8312 REF=PVl.s8312[HMI.HMI_8312_Index];	
	s8312_mapping.PT_203:	GW_TK201.Node:=PVl.s8312[HMI.HMI_8312_Index].DSO.Node; GW_TK201.r8312 REF=PVl.s8312[HMI.HMI_8312_Index];
	


	
END_CASE;
              
END_ACTION

ACTION ME44AI_Select:
                CASE HMI.HMI_ME44AI_Index OF
	
	ME44AI_Mapping.GW100_S2:	GW_Z100.rME44AI REF= Network.ME44_AI[HMI.HMI_ME44AI_Index];
								GW_Z100.Node:=	Network.ME44_AI[HMI.HMI_ME44AI_Index].DSO.Node;
								
	ME44AI_Mapping.GW100_S3:	GW_Z100.rME44AI REF= Network.ME44_AI[HMI.HMI_ME44AI_Index];
								GW_Z100.Node:=	Network.ME44_AI[HMI.HMI_ME44AI_Index].DSO.Node;
								
	ME44AI_Mapping.GW201_S2:	GW_Z201.rME44AI REF= Network.ME44_AI[HMI.HMI_ME44AI_Index];
								GW_Z201.Node:=	Network.ME44_AI[HMI.HMI_ME44AI_Index].DSO.Node;
								
	ME44AI_Mapping.GW202_S3:	GW_Z202.rME44AI REF= Network.ME44_AI[HMI.HMI_ME44AI_Index];
								GW_Z202.Node:=	Network.ME44_AI[HMI.HMI_ME44AI_Index].DSO.Node;
								
								
								
								
								
	(*
	4:	GW_Branch_1.Node:=Network.Branch_1_ME44_S4_AI.DSO.Node; GW_Branch_1.rME44AI REF=Network.Branch_1_ME44_S4_AI; Burkert.HMI_ME44AI_Sync(Local:=Network.Branch_1_ME44_S4_AI,HMI:=HMI.HMI_ME44AI_data);
	5:	GW_Branch_2.Node:=Network.Branch_2_ME44_S4_AI.DSO.Node; GW_Branch_2.rME44AI REF=Network.Branch_2_ME44_S4_AI; Burkert.HMI_ME44AI_Sync(Local:=Network.Branch_2_ME44_S4_AI,HMI:=HMI.HMI_ME44AI_data);
	6:	GW_Branch_3.Node:=Network.Branch_3_ME44_S4_AI.DSO.Node; GW_Branch_3.rME44AI REF=Network.Branch_3_ME44_S4_AI; Burkert.HMI_ME44AI_Sync(Local:=Network.Branch_3_ME44_S4_AI,HMI:=HMI.HMI_ME44AI_data);
	7:	GW_Branch_4.Node:=Network.Branch_4_ME44_S4_AI.DSO.Node; GW_Branch_4.rME44AI REF=Network.Branch_4_ME44_S4_AI; Burkert.HMI_ME44AI_Sync(Local:=Network.Branch_4_ME44_S4_AI,HMI:=HMI.HMI_ME44AI_data);
	8:	GW_Branch_5.Node:=Network.Branch_5_ME44_S4_AI.DSO.Node; GW_Branch_5.rME44AI REF=Network.Branch_5_ME44_S4_AI; Burkert.HMI_ME44AI_Sync(Local:=Network.Branch_5_ME44_S4_AI,HMI:=HMI.HMI_ME44AI_data);
	9:	
		GW_Branch_6.Node:=Network.Branch_6_ME44_S4_AI.DSO.Node; 
		GW_Branch_6.rME44AI REF=Network.Branch_6_ME44_S4_AI; 
		Burkert.HMI_ME44AI_Sync(Local:=Network.Branch_6_ME44_S4_AI,HMI:=HMI.HMI_ME44AI_data);
	*)
END_CASE
              
END_ACTION

ACTION s336x_Select:
                CASE HMI.HMI_336x_Index OF
	s3363_mapping.ACV_101:	GW_Z100.Node:=GVL.s3363[HMI.HMI_336x_Index].DSO.Node; GW_Z100.r336x REF=GVl.s3363[HMI.HMI_336x_Index];
	s3363_mapping.ACV_102:	GW_Z100.Node:=GVL.s3363[HMI.HMI_336x_Index].DSO.Node; GW_Z100.r336x REF=GVl.s3363[HMI.HMI_336x_Index];
	
END_CASE
              
END_ACTION

ACTION ACV_Select:
                
CASE HMI.HMI_ACV_Index OF
	

	(*
	ACV_Mapping.Branch_1_CW1:			GW_Branch_1.r8694 REF= GVL.ACV[ACV_Mapping.Branch_1_CW1]; 		Gw_branch_1.Node:=GVL.ACV[ACV_Mapping.Branch_1_CW1].DSO.Node; 
	ACV_Mapping.Branch_1_CW2:			GW_Branch_1.r8694 REF= GVL.ACV[ACV_Mapping.Branch_1_CW2]; 		Gw_branch_1.Node:=GVL.ACV[ACV_Mapping.Branch_1_CW2].DSO.Node;
	ACV_Mapping.Branch_1_HW1:			GW_Branch_1.r8694 REF= GVL.ACV[ACV_Mapping.Branch_1_HW1]; 		Gw_branch_1.Node:=GVL.ACV[ACV_Mapping.Branch_1_HW1].DSO.Node;
	ACV_Mapping.Branch_1_HW2:			GW_Branch_1.r8694 REF= GVL.ACV[ACV_Mapping.Branch_1_HW2]; 		GW_branch_1.Node:=GVL.ACV[ACV_Mapping.Branch_1_HW2].DSO.Node;
	ACV_Mapping.Branch_1_Discharge :	GW_Branch_1.r8694 REF= GVL.ACV[ACV_Mapping.Branch_1_Discharge]; Gw_branch_1.Node:=GVL.ACV[ACV_Mapping.Branch_1_Discharge].DSO.Node; 
	
	ACV_Mapping.Branch_2_CW1:			GW_Branch_2.r8694 REF= GVL.ACV[ACV_Mapping.Branch_2_CW1]; 		Gw_branch_2.Node:=GVL.ACV[ACV_Mapping.Branch_2_CW1].DSO.Node; 
	ACV_Mapping.Branch_2_CW2:			GW_Branch_2.r8694 REF= GVL.ACV[ACV_Mapping.Branch_2_CW2]; 		Gw_branch_2.Node:=GVL.ACV[ACV_Mapping.Branch_2_CW2].DSO.Node;
	ACV_Mapping.Branch_2_HW1:			GW_Branch_2.r8694 REF= GVL.ACV[ACV_Mapping.Branch_2_HW1]; 		Gw_branch_2.Node:=GVL.ACV[ACV_Mapping.Branch_2_HW1].DSO.Node;
	ACV_Mapping.Branch_2_HW2:			GW_Branch_2.r8694 REF= GVL.ACV[ACV_Mapping.Branch_2_HW2]; 		GW_branch_2.Node:=GVL.ACV[ACV_Mapping.Branch_2_HW2].DSO.Node;
	ACV_Mapping.Branch_2_Discharge :	GW_Branch_2.r8694 REF= GVL.ACV[ACV_Mapping.Branch_2_Discharge]; Gw_branch_2.Node:=GVL.ACV[ACV_Mapping.Branch_2_Discharge].DSO.Node; 
	
	ACV_Mapping.Branch_3_CW1:			GW_Branch_3.r8694 REF= GVL.ACV[ACV_Mapping.Branch_3_CW1]; 		Gw_branch_3.Node:=GVL.ACV[ACV_Mapping.Branch_3_CW1].DSO.Node; 
	ACV_Mapping.Branch_3_CW2:			GW_Branch_3.r8694 REF= GVL.ACV[ACV_Mapping.Branch_3_CW2]; 		Gw_branch_3.Node:=GVL.ACV[ACV_Mapping.Branch_3_CW2].DSO.Node;
	ACV_Mapping.Branch_3_HW1:			GW_Branch_3.r8694 REF= GVL.ACV[ACV_Mapping.Branch_3_HW1]; 		Gw_branch_3.Node:=GVL.ACV[ACV_Mapping.Branch_3_HW1].DSO.Node;
	ACV_Mapping.Branch_3_HW2:			GW_Branch_3.r8694 REF= GVL.ACV[ACV_Mapping.Branch_3_HW2]; 		GW_branch_3.Node:=GVL.ACV[ACV_Mapping.Branch_3_HW2].DSO.Node;
	ACV_Mapping.Branch_3_Discharge :	GW_Branch_3.r8694 REF= GVL.ACV[ACV_Mapping.Branch_3_Discharge]; Gw_branch_3.Node:=GVL.ACV[ACV_Mapping.Branch_3_Discharge].DSO.Node; 
	
	ACV_Mapping.Branch_4_CW1:			GW_Branch_4.r8694 REF= GVL.ACV[ACV_Mapping.Branch_4_CW1]; 		Gw_branch_4.Node:=GVL.ACV[ACV_Mapping.Branch_4_CW1].DSO.Node; 
	ACV_Mapping.Branch_4_CW2:			GW_Branch_4.r8694 REF= GVL.ACV[ACV_Mapping.Branch_4_CW2]; 		Gw_branch_4.Node:=GVL.ACV[ACV_Mapping.Branch_4_CW2].DSO.Node;
	ACV_Mapping.Branch_4_HW1:			GW_Branch_4.r8694 REF= GVL.ACV[ACV_Mapping.Branch_4_HW1]; 		Gw_branch_4.Node:=GVL.ACV[ACV_Mapping.Branch_4_HW1].DSO.Node;
	ACV_Mapping.Branch_4_HW2:			GW_Branch_4.r8694 REF= GVL.ACV[ACV_Mapping.Branch_4_HW2]; 		GW_branch_4.Node:=GVL.ACV[ACV_Mapping.Branch_4_HW2].DSO.Node;
	ACV_Mapping.Branch_4_Discharge :	GW_Branch_4.r8694 REF= GVL.ACV[ACV_Mapping.Branch_4_Discharge]; Gw_branch_4.Node:=GVL.ACV[ACV_Mapping.Branch_4_Discharge].DSO.Node; 
	
	ACV_Mapping.Branch_5_CW1:			GW_Branch_5.r8694 REF= GVL.ACV[ACV_Mapping.Branch_5_CW1]; 				Gw_branch_5.Node:=GVL.ACV[ACV_Mapping.Branch_5_CW1].DSO.Node; 
	ACV_Mapping.Branch_5_CW2:			GW_Branch_5.r8694 REF= GVL.ACV[ACV_Mapping.Branch_5_CW2]; 				Gw_branch_5.Node:=GVL.ACV[ACV_Mapping.Branch_5_CW2].DSO.Node;
	ACV_Mapping.Branch_5_HW1:			GW_Branch_5.r8694 REF= GVL.ACV[ACV_Mapping.Branch_5_HW1]; 				Gw_branch_5.Node:=GVL.ACV[ACV_Mapping.Branch_5_HW1].DSO.Node;
	ACV_Mapping.Branch_5_HW2:			GW_Branch_5.r8694 REF= GVL.ACV[ACV_Mapping.Branch_5_HW2]; 				GW_branch_5.Node:=GVL.ACV[ACV_Mapping.Branch_5_HW2].DSO.Node;
	ACV_Mapping.Branch_5_Discharge :	GW_Branch_5.r8694 REF= GVL.ACV[ACV_Mapping.Branch_5_Discharge]; 		Gw_branch_5.Node:=GVL.ACV[ACV_Mapping.Branch_5_Discharge].DSO.Node; 
	
	ACV_Mapping.ALS_Cold_Water_Return_Valve:			GW_CWS.r8694 REF= GVL.ACV[ACV_Mapping.ALS_Cold_Water_Return_Valve]; 				Gw_CWS.Node:=GVL.ACV[ACV_Mapping.ALS_Cold_Water_Return_Valve].DSO.Node; 
	ACV_MApping.ALS_Hot_Water_Return_Valve:				GW_HWS.r8694 REF= GVL.ACV[ACV_Mapping.ALS_Hot_Water_Return_Valve]; 					Gw_HWS.Node:=GVL.ACV[ACV_Mapping.ALS_Hot_Water_Return_Valve].DSO.Node; 
	ACV_Mapping.E201_Circulation_Water_Supply_Valve:	GW_CWS.r8694 REF= GVL.ACV[ACV_Mapping.E201_Circulation_Water_Supply_Valve]; 	Gw_CWS.Node:=GVL.ACV[ACV_Mapping.E201_Circulation_Water_Supply_Valve].DSO.Node; 
	ACV_MApping.E201_Glycol_Supply_Valve:				GW_CWS.r8694 REF= GVL.ACV[ACV_Mapping.E201_Glycol_Supply_Valve]; 				Gw_CWS.Node:=GVL.ACV[ACV_Mapping.E201_Glycol_Supply_Valve].DSO.Node; 
	ACV_Mapping.H202_Circulation_Water_Supply_Valve:	GW_HWS.r8694 REF= GVL.ACV[ACV_Mapping.H202_Circulation_Water_Supply_Valve]; 	Gw_HWS.Node:=GVL.ACV[ACV_Mapping.H202_Circulation_Water_Supply_Valve].DSO.Node; 
	ACV_MApping.TK201_RO_MakeUp_Flow_Valve:				GW_CWS.r8694 REF= GVL.ACV[ACV_Mapping.TK201_RO_MakeUp_Flow_Valve]; 				Gw_CWS.Node:=GVL.ACV[ACV_Mapping.TK201_RO_MakeUp_Flow_Valve].DSO.Node; 
	ACV_Mapping.TK202_RO_MakeUp_Flow_Valve:				GW_HWS.r8694 REF= GVL.ACV[ACV_Mapping.TK202_RO_MakeUp_Flow_Valve]; 				Gw_HWS.Node:=GVL.ACV[ACV_Mapping.TK202_RO_MakeUp_Flow_Valve].DSO.Node; 
	

*)
END_CASE

              
END_ACTION

ACTION pm8653_Select:
                CASE HMI.HMI_8653_Index OF
(*
	11	:	GW_CWS.Node:=11;		GW_CWS.r8653 REF= Network.CWS_PM5; 			Burkert.HMI_8653_Sync(Local:=Network.CWS_PM5,HMI:=HMI.HMI_8653_data);
	20	:	GW_HWS.Node:=20;		GW_HWS.r8653 REF= Network.HWS_PM4;			Burkert.HMI_8653_Sync(Local:=Network.HWS_PM4,HMI:=HMI.HMI_8653_data);
	26	:	GW_Ro.Node:=26;			GW_Ro.r8653 REF= Network.RO_PM3;			Burkert.HMI_8653_Sync(Local:=Network.Ro_PM3,HMI:=HMI.HMI_8653_data);
	40	: 	GW_Branch_1.Node:=40;	GW_Branch_1.r8653 REF= Network.Branch_1_PM;	Burkert.HMI_8653_Sync(Local:=Network.Branch_1_PM,HMI:=HMI.HMI_8653_data);
	55 	: 	GW_Branch_2.Node:=55;	GW_Branch_2.r8653 REF= Network.Branch_2_PM;	Burkert.HMI_8653_Sync(Local:=Network.Branch_2_PM,HMI:=HMI.HMI_8653_data);
	70	:	GW_Branch_3.Node:=70;	GW_Branch_3.r8653 REF= Network.Branch_3_PM;	Burkert.HMI_8653_Sync(Local:=Network.Branch_3_PM,HMI:=HMI.HMI_8653_data);
	85	:	GW_Branch_4.Node:=85;	GW_Branch_4.r8653 REF= Network.Branch_4_PM;	Burkert.HMI_8653_Sync(Local:=Network.Branch_4_PM,HMI:=HMI.HMI_8653_data);
	100	:	GW_Branch_5.Node:=100;	GW_Branch_5.r8653 REF= Network.Branch_5_PM;	Burkert.HMI_8653_Sync(Local:=Network.Branch_5_PM,HMI:=HMI.HMI_8653_data);
	125	:	GW_Branch_6.Node:=125;	GW_Branch_6.r8653 REF= Network.Branch_6_PM;	Burkert.HMI_8653_Sync(Local:=Network.Branch_6_PM,HMI:=HMI.HMI_8653_data);
	
*)		
END_CASE
              
END_ACTION
END_PROGRAM

PROGRAM s8228_Manager
  VAR
    CT_122_CTRL : Burkert.CanOpen_8228;
    CT_131_CTRL : Burkert.CanOpen_8228;
    CT_142_CTRL : Burkert.CanOpen_8228;
  END_VAR

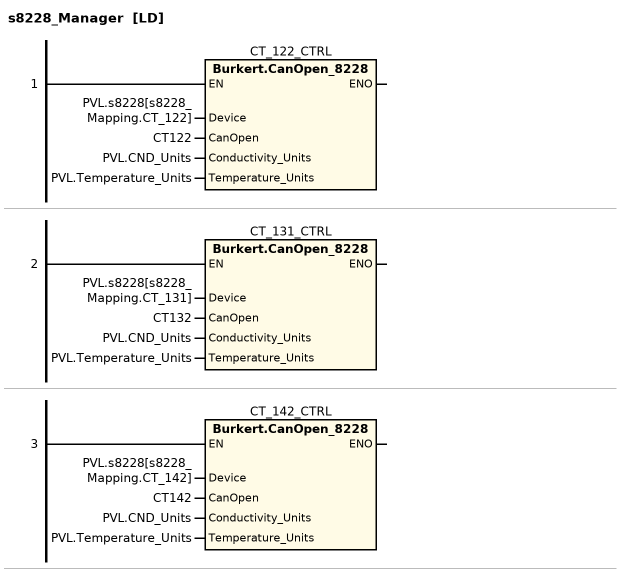
(* LD diagram, written out as Structured Text *)

CT_122_CTRL(Device := PVL.s8228[s8228_Mapping.CT_122], CanOpen := CT122, Conductivity_Units := PVL.CND_Units, Temperature_Units := PVL.Temperature_Units);

CT_131_CTRL(Device := PVL.s8228[s8228_Mapping.CT_131], CanOpen := CT132, Conductivity_Units := PVL.CND_Units, Temperature_Units := PVL.Temperature_Units);

CT_142_CTRL(Device := PVL.s8228[s8228_Mapping.CT_142], CanOpen := CT142, Conductivity_Units := PVL.CND_Units, Temperature_Units := PVL.Temperature_Units);
END_PROGRAM

PROGRAM AIT_Manager
  VAR
    LT_101_P_CTRL : Burkert.Analog_Sensor_UDFB;
    LT_201_CTRL : Burkert.Analog_Sensor_UDFB;
    LT_201A_P_CTRL : Burkert.Analog_Sensor_UDFB;
    LT_202_CTRL : Burkert.Analog_Sensor_UDFB;
    LT_202A_CTRL : Burkert.Analog_Sensor_UDFB;
    LT_001_CTRL : Burkert.Analog_Sensor_UDFB;
    LT_002_CTRL : Burkert.Analog_Sensor_UDFB;
    UV_001_CTRL : Burkert.Analog_Sensor_UDFB;
    FT_01_CTRL : Burkert.Analog_Sensor_UDFB;
  END_VAR

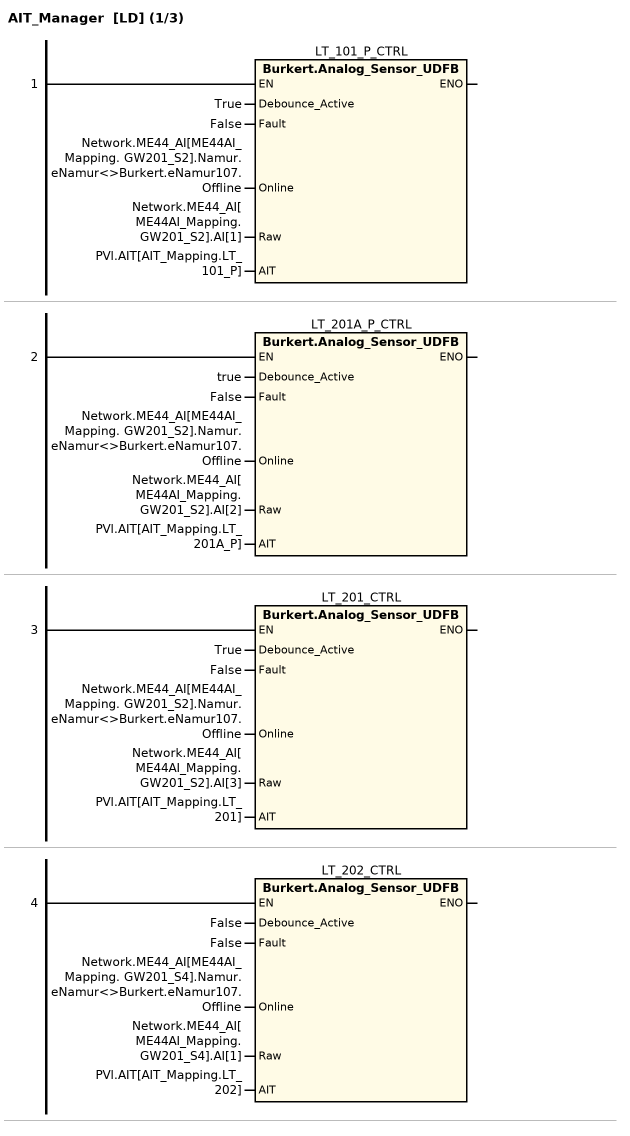
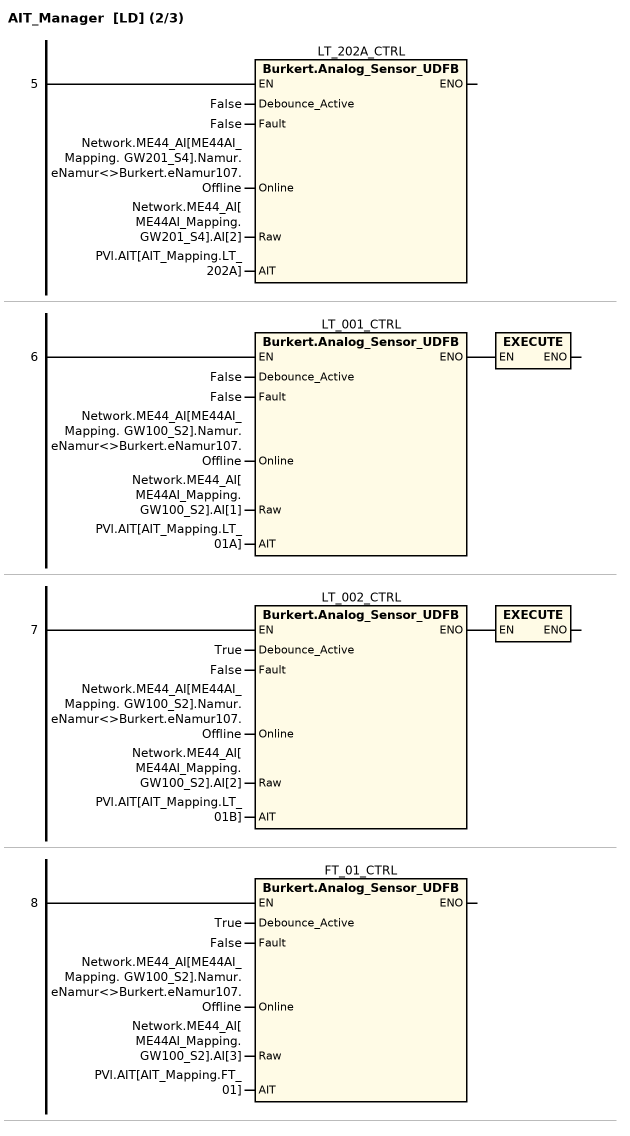
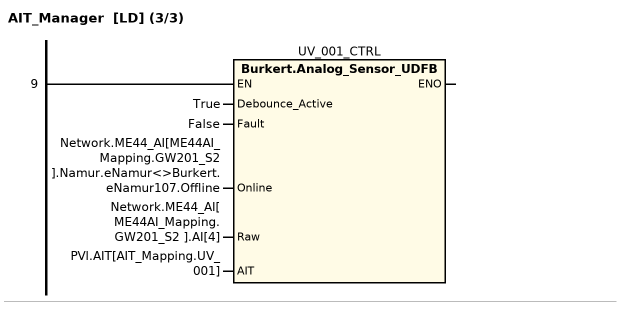
(* LD diagram, written out as Structured Text *)

LT_101_P_CTRL(Debounce_Active := True, Fault := False, Online := Network.ME44_AI[ME44AI_Mapping. GW201_S2].Namur.eNamur<>Burkert.eNamur107.Offline, Raw := Network.ME44_AI[ME44AI_Mapping. GW201_S2].AI[1], AIT := PVl.AIT[AIT_Mapping.LT_101_P]);


LT_201A_P_CTRL(Debounce_Active := true, Fault := False, Online := Network.ME44_AI[ME44AI_Mapping. GW201_S2].Namur.eNamur<>Burkert.eNamur107.Offline, Raw := Network.ME44_AI[ME44AI_Mapping. GW201_S2].AI[2], AIT := PVl.AIT[AIT_Mapping.LT_201A_P]);

LT_201_CTRL(Debounce_Active := True, Fault := False, Online := Network.ME44_AI[ME44AI_Mapping. GW201_S2].Namur.eNamur<>Burkert.eNamur107.Offline, Raw := Network.ME44_AI[ME44AI_Mapping. GW201_S2].AI[3], AIT := PVl.AIT[AIT_Mapping.LT_201]);

LT_202_CTRL(Debounce_Active := False, Fault := False, Online := Network.ME44_AI[ME44AI_Mapping. GW201_S4].Namur.eNamur<>Burkert.eNamur107.Offline, Raw := Network.ME44_AI[ME44AI_Mapping. GW201_S4].AI[1], AIT := PVl.AIT[AIT_Mapping.LT_202]);

LT_202A_CTRL(Debounce_Active := False, Fault := False, Online := Network.ME44_AI[ME44AI_Mapping. GW201_S4].Namur.eNamur<>Burkert.eNamur107.Offline, Raw := Network.ME44_AI[ME44AI_Mapping. GW201_S4].AI[2], AIT := PVl.AIT[AIT_Mapping.LT_202A]);

LT_001_CTRL(Debounce_Active := False, Fault := False, Online := Network.ME44_AI[ME44AI_Mapping. GW100_S2].Namur.eNamur<>Burkert.eNamur107.Offline, Raw := Network.ME44_AI[ME44AI_Mapping. GW100_S2].AI[1], AIT := PVl.AIT[AIT_Mapping.LT_01A]);
IF LT_001_CTRL.ENO THEN
  PVl.AIT[AIT_Mapping.LT_01A].Alarm_Config.Silence:=True;
END_IF;

LT_002_CTRL(Debounce_Active := True, Fault := False, Online := Network.ME44_AI[ME44AI_Mapping. GW100_S2].Namur.eNamur<>Burkert.eNamur107.Offline, Raw := Network.ME44_AI[ME44AI_Mapping. GW100_S2].AI[2], AIT := PVl.AIT[AIT_Mapping.LT_01B]);
IF LT_002_CTRL.ENO THEN
  PVl.AIT[AIT_Mapping.LT_01B].Alarm_Config.Silence:=TRUE;
END_IF;

FT_01_CTRL(Debounce_Active := True, Fault := False, Online := Network.ME44_AI[ME44AI_Mapping. GW100_S2].Namur.eNamur<>Burkert.eNamur107.Offline, Raw := Network.ME44_AI[ME44AI_Mapping. GW100_S2].AI[3], AIT := PVl.AIT[AIT_Mapping.FT_01]);

UV_001_CTRL(Debounce_Active := True, Fault := False, Online := Network.ME44_AI[ME44AI_Mapping.GW201_S2 ].Namur.eNamur<>Burkert.eNamur107.Offline, Raw := Network.ME44_AI[ME44AI_Mapping.GW201_S2 ].AI[4], AIT := PVl.AIT[AIT_Mapping.UV_001]);
END_PROGRAM

PROGRAM Adam_6250

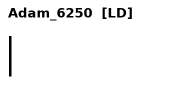
(* LD diagram, written out as Structured Text *)
END_PROGRAM

PROGRAM Level_1_CTRL

            FIT_Manager();
Flowave_manager();
s336x_manager();
PT_Manager();
LS_Manager();
VFD_Manager();
BCV_Manager();
AIT_Manager();
DO_Manager();
DI_Manager();







          
END_PROGRAM

PROGRAM Filter_Manager
  VAR
    Filter_1 : Burkert.fb_ACV_Filter;
    tACV : Burkert.cACV;
    Filter_204B : Burkert.fb_ACV_Filter;
    Filter_205A : Burkert.fb_ACV_Filter;
    Filter_205B : Burkert.fb_ACV_Filter;
    Filters_204 : Burkert.Filter_Pair;
    Filters_205 : Burkert.Filter_Pair;
    Bypass_rTrig : r_Trig;
    Auto_rTrig : R_TRIG;
    Off_rTrig : R_TRIG;
    Prime_SR_0 : SR;
    Manual_rTrig : R_TRIG;
    TOF_0 : TOF;
    TP_0 : TP;
  END_VAR
  VAR  (* added by the conversion: wires and edge detectors of the diagram *)
    _SEL6_OUT : ANY;
    _SEL2_OUT : ANY;
    _SEL37_OUT : ANY;
    _SEL14_OUT : ANY;
    _SEL54_OUT : ANY;
    _OR8_OUT : BOOL;
    _OR43_OUT : BOOL;
    _SEL54_OUT_2 : BOOL;
    _AND46_OUT : BOOL;
    _SEL76_OUT : ANY;
  END_VAR

            
tACV.ready:=TRUE;

Alarms();
Aux();
modes();
Bypass_Valve_CTRL();
Evaluate_All();
Filter_CTRL();

//GVL.s3363[s3363_mapping.ACV_219].PLC_CMD:=SEL(	( PVL.Filters[0].Mode.eMode=Burkert.eFilter_Manager_Modes.Disabled AND PVL.Filters[1].Mode.eMode=Burkert.eFilter_Manager_Modes.Disabled),0,100);

IF (
	PVl.Filters[0].Mode.eMode=Burkert.eFilter_Manager_Modes.Filter_1 OR
	PVl.Filters[0].Mode.eMode=Burkert.eFilter_Manager_Modes.Filter_2 OR
	PVl.Filters[1].Mode.eMode=Burkert.eFilter_Manager_Modes.Filter_1 OR
	PVl.Filters[1].Mode.eMode=Burkert.eFilter_Manager_Modes.Filter_2 OR
	(PVl.Filters[0].Mode.eMode=Burkert.eFilter_Manager_Modes.Disabled AND PVL.Filter_Config.Mode.eMode=eFilter_mode.Auto) OR
	(PVl.Filters[1].Mode.eMode=Burkert.eFilter_Manager_Modes.Disabled AND PVL.Filter_Config.Mode.eMode=eFilter_mode.Auto) ) THEN
	PVL.Filter_Config.Mode.eMode:=eFilter_mode.Manual;
END_IF;

	
          

ACTION Aux:
                PVL.filter_Config.StrMode:=Burkert.Burkert_OSCAT_BASIC.REPLACE_ALL(str:=TO_STRING(PVL.Filter_Config.Mode.eMode) , src:='_' , rep:=' ' );
PVL.Filter_Config.StrStatus:=Burkert.Burkert_OSCAT_BASIC.REPLACE_ALL(str:=TO_STRING(PVL.Filter_Config.Status.eStatus) , src:='_' , rep:=' ' );

PVL.filters[0].DP.EU:=PVl.s8312[s8312_Mapping.PT_202].EU-PVl.s8312[s8312_Mapping.PT_204].EU;
PVL.filters[1].DP.EU:=PVl.s8312[s8312_Mapping.PT_204].EU-PVl.s8312[s8312_Mapping.PT_205].EU;


GVL.Filter_Path_Available:=(
	GVL.s3363[s3363_Mapping.ACV_219].Valve_Actual>10 OR
	(
		(PVl.Filters[0].Filter_1.Status.eStatus=Burkert.eFilter_Status.In_Service OR PVl.Filters[0].Filter_2.Status.eStatus=Burkert.eFilter_Status.In_Service) AND
		(PVl.Filters[1].Filter_1.Status.eStatus=Burkert.eFilter_Status.In_Service OR PVl.Filters[1].Filter_2.Status.eStatus=Burkert.eFilter_Status.In_Service))
	);
	
	


              
END_ACTION

ACTION Filter_CTRL:
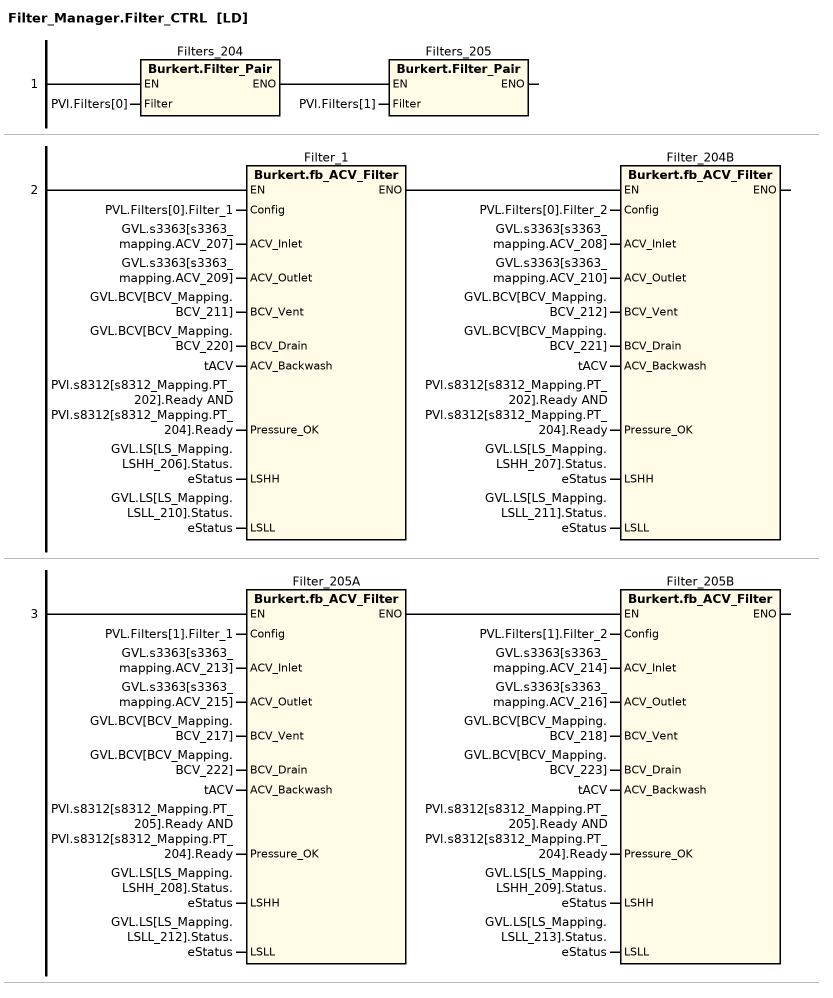
(* LD diagram, written out as Structured Text *)

Filters_204(Filter := PVl.Filters[0]);
Filters_205(EN := Filters_204.ENO, Filter := PVl.Filters[1]);

Filter_1(Config := PVL.Filters[0].Filter_1, ACV_Inlet := GVL.s3363[s3363_mapping.ACV_207], ACV_Outlet := GVL.s3363[s3363_mapping.ACV_209], BCV_Vent := GVL.BCV[BCV_Mapping.BCV_211], BCV_Drain := GVL.BCV[BCV_Mapping.BCV_220], ACV_Backwash := tACV, Pressure_OK := PVl.s8312[s8312_Mapping.PT_202].Ready AND PVl.s8312[s8312_Mapping.PT_204].Ready, LSHH := GVL.LS[LS_Mapping.LSHH_206].Status.eStatus, LSLL := GVL.LS[LS_Mapping.LSLL_210].Status.eStatus);
Filter_204B(EN := Filter_1.ENO, Config := PVL.Filters[0].Filter_2, ACV_Inlet := GVL.s3363[s3363_mapping.ACV_208], ACV_Outlet := GVL.s3363[s3363_mapping.ACV_210], BCV_Vent := GVL.BCV[BCV_Mapping.BCV_212], BCV_Drain := GVL.BCV[BCV_Mapping.BCV_221], ACV_Backwash := tACV, Pressure_OK := PVl.s8312[s8312_Mapping.PT_202].Ready AND PVl.s8312[s8312_Mapping.PT_204].Ready, LSHH := GVL.LS[LS_Mapping.LSHH_207].Status.eStatus, LSLL := GVL.LS[LS_Mapping.LSLL_211].Status.eStatus);

Filter_205A(Config := PVL.Filters[1].Filter_1, ACV_Inlet := GVL.s3363[s3363_mapping.ACV_213], ACV_Outlet := GVL.s3363[s3363_mapping.ACV_215], BCV_Vent := GVL.BCV[BCV_Mapping.BCV_217], BCV_Drain := GVL.BCV[BCV_Mapping.BCV_222], ACV_Backwash := tACV, Pressure_OK := PVl.s8312[s8312_Mapping.PT_205].Ready AND PVl.s8312[s8312_Mapping.PT_204].Ready, LSHH := GVL.LS[LS_Mapping.LSHH_208].Status.eStatus, LSLL := GVL.LS[LS_Mapping.LSLL_212].Status.eStatus);
Filter_205B(EN := Filter_205A.ENO, Config := PVL.Filters[1].Filter_2, ACV_Inlet := GVL.s3363[s3363_mapping.ACV_214], ACV_Outlet := GVL.s3363[s3363_mapping.ACV_216], BCV_Vent := GVL.BCV[BCV_Mapping.BCV_218], BCV_Drain := GVL.BCV[BCV_Mapping.BCV_223], ACV_Backwash := tACV, Pressure_OK := PVl.s8312[s8312_Mapping.PT_205].Ready AND PVl.s8312[s8312_Mapping.PT_204].Ready, LSHH := GVL.LS[LS_Mapping.LSHH_209].Status.eStatus, LSLL := GVL.LS[LS_Mapping.LSLL_213].Status.eStatus);
(* --- network --- *)
END_ACTION

ACTION Alarms:
                (*PVL.Filters[0].DP.Alarm_Config.Low_Low_Alarm:=(-1);
PVL.Filters[0].DP.Alarm_Config.Low_Warn:=(-0.9);
PVL.Filters[0].DP.Alarm_Config.Low_Norm:=(-0.8);
PVL.Filters[0].DP.Alarm_Config.Hi_Norm:=PVL.Filters[0].DP.Alarm_Config.Hi_Hi_Alarm-0.02;
PVL.Filters[0].DP.Alarm_Config.Hi_Warn:=PVL.Filters[0].DP.Alarm_Config.Hi_Hi_Alarm-0.01;
PVL.Filters[0].DP.Alarm_Config.Debounce:=1;
*)
PVL.Filters[0].DP.Alarm_Config.Silence:=NOT(PVL.Filter_Config.Mode.eMode=eFilter_Mode.Manual OR PVL.Filter_Config.Mode.eMode=eFilter_Mode.Auto)	;
(*
PVL.Filters[1].DP.Alarm_Config.Low_Low_Alarm:=(-1);
PVL.Filters[1].DP.Alarm_Config.Low_Warn:=(-0.9);
PVL.Filters[1].DP.Alarm_Config.Low_Norm:=(-0.8);
PVL.Filters[1].DP.Alarm_Config.Hi_Norm:=PVL.Filters[0].DP.Alarm_Config.Hi_Hi_Alarm-0.02;
PVL.Filters[1].DP.Alarm_Config.Hi_Warn:=PVL.Filters[0].DP.Alarm_Config.Hi_Hi_Alarm-0.01;
PVL.Filters[1].DP.Alarm_Config.Debounce:=1;
*)
PVL.Filters[1].DP.Alarm_Config.Silence:=NOT(PVL.Filter_Config.Mode.eMode=eFilter_Mode.Manual OR PVL.Filter_Config.Mode.eMode=eFilter_Mode.Auto);


(*
PVl.s8312[S8312_mapping.PT_202].Alarm_Config.Silence:=	PVl.Filter_Config.Mode.eMode=eFilter_Mode.Off;

PVl.s8098[s8098_Mapping.FT_202].PDO.VolumeFlow .Alarm_Config.Silence:=	PVl.Filter_Config.Mode.eMode=eFilter_Mode.Off;
PVl.s8098[s8098_Mapping.FT_202].PDO.Totaliser_1 .Alarm_Config.Silence:=	PVl.Filter_Config.Mode.eMode=eFilter_Mode.Off;

*)

PVl.s8098[s8098_Mapping.FT_204].PDO.VolumeFlow .Alarm_Config.Silence:=	PVl.Filter_Config.Mode.eMode=eFilter_Mode.Off;
PVl.s8098[s8098_Mapping.FT_204].PDO.Totaliser_1 .Alarm_Config.Silence:=	PVl.Filter_Config.Mode.eMode=eFilter_Mode.Off;
PVl.s8312[S8312_mapping.PT_204].Alarm_Config.Silence:=	PVl.Filter_Config.Mode.eMode=eFilter_Mode.Off;
PVl.s8312[S8312_mapping.PT_205].Alarm_Config.Silence:=	PVl.Filter_Config.Mode.eMode=eFilter_Mode.Off;


PVL.s8098[s8098_mapping.FT_204].PDO.VolumeFlow.Alarm_Config:=PVL.s8098[s8098_mapping.FT_202].PDO.VolumeFlow.Alarm_Config;
PVL.s8098[s8098_mapping.FT_204].PDO.Totaliser_1.Alarm_Config.Silence:=FALSE;

PVl.s8312[s8312_Mapping.PT_205].Alarm_Config.Low_Low_Alarm:=(-5.0);
PVl.s8312[s8312_Mapping.PT_205].Alarm_Config.Low_warn:=(-4);

PVl.s8312[s8312_Mapping.PT_202].Alarm_Config.Low_Low_Alarm:=(-5.0);
PVl.s8312[s8312_Mapping.PT_202].Alarm_Config.Low_warn:=(-4);


PVl.s8312[s8312_Mapping.PT_204].Alarm_Config.Low_Low_Alarm:=(-5.0);
PVl.s8312[s8312_Mapping.PT_204].Alarm_Config.Low_warn:=(-4);


 
              
END_ACTION

ACTION Modes:
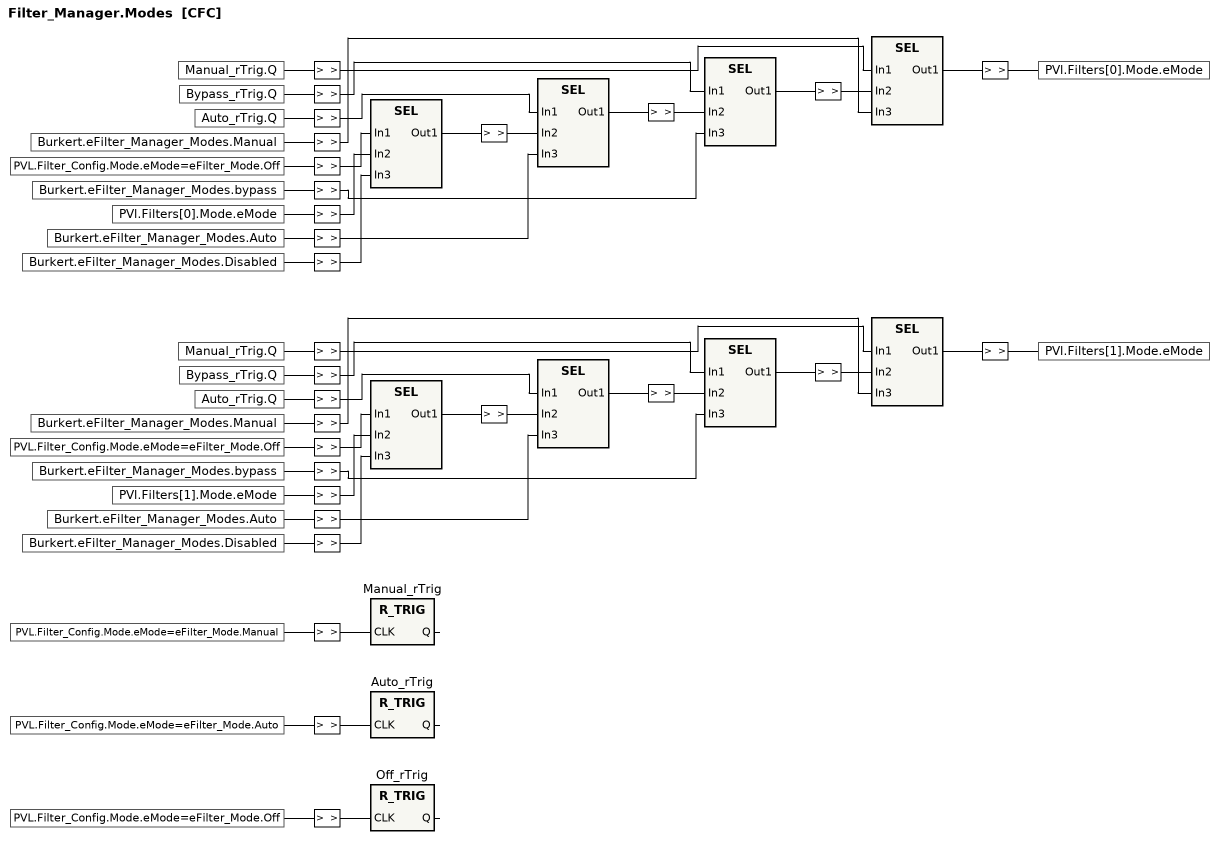
(* CFC diagram, written out as Structured Text *)
_SEL2_OUT := SEL(Manual_rTrig.Q, _SEL6_OUT, Burkert.eFilter_Manager_Modes.Manual);
Manual_rTrig(CLK := PVL.Filter_Config.Mode.eMode=eFilter_Mode.Manual);
Auto_rTrig(CLK := PVL.Filter_Config.Mode.eMode=eFilter_Mode.Auto);
_SEL6_OUT := SEL(Bypass_rTrig.Q, SEL(Auto_rTrig.Q, _SEL14_OUT, Burkert.eFilter_Manager_Modes.Auto), Burkert.eFilter_Manager_Modes.bypass);
PVl.Filters[1].Mode.eMode := _SEL2_OUT;
Off_rTrig(CLK := PVL.Filter_Config.Mode.eMode=eFilter_Mode.Off);
_SEL37_OUT := SEL(PVL.Filter_Config.Mode.eMode=eFilter_Mode.Off, PVl.Filters[0].Mode.eMode, Burkert.eFilter_Manager_Modes.Disabled);
_SEL14_OUT := SEL(PVL.Filter_Config.Mode.eMode=eFilter_Mode.Off, PVl.Filters[1].Mode.eMode, Burkert.eFilter_Manager_Modes.Disabled);
_SEL54_OUT := SEL(Bypass_rTrig.Q, SEL(Auto_rTrig.Q, _SEL37_OUT, Burkert.eFilter_Manager_Modes.Auto), Burkert.eFilter_Manager_Modes.bypass);
PVl.Filters[0].Mode.eMode := SEL(Manual_rTrig.Q, _SEL54_OUT, Burkert.eFilter_Manager_Modes.Manual);
END_ACTION

ACTION Evaluate_All:
                
              
END_ACTION

ACTION Bypass_Valve_CTRL:
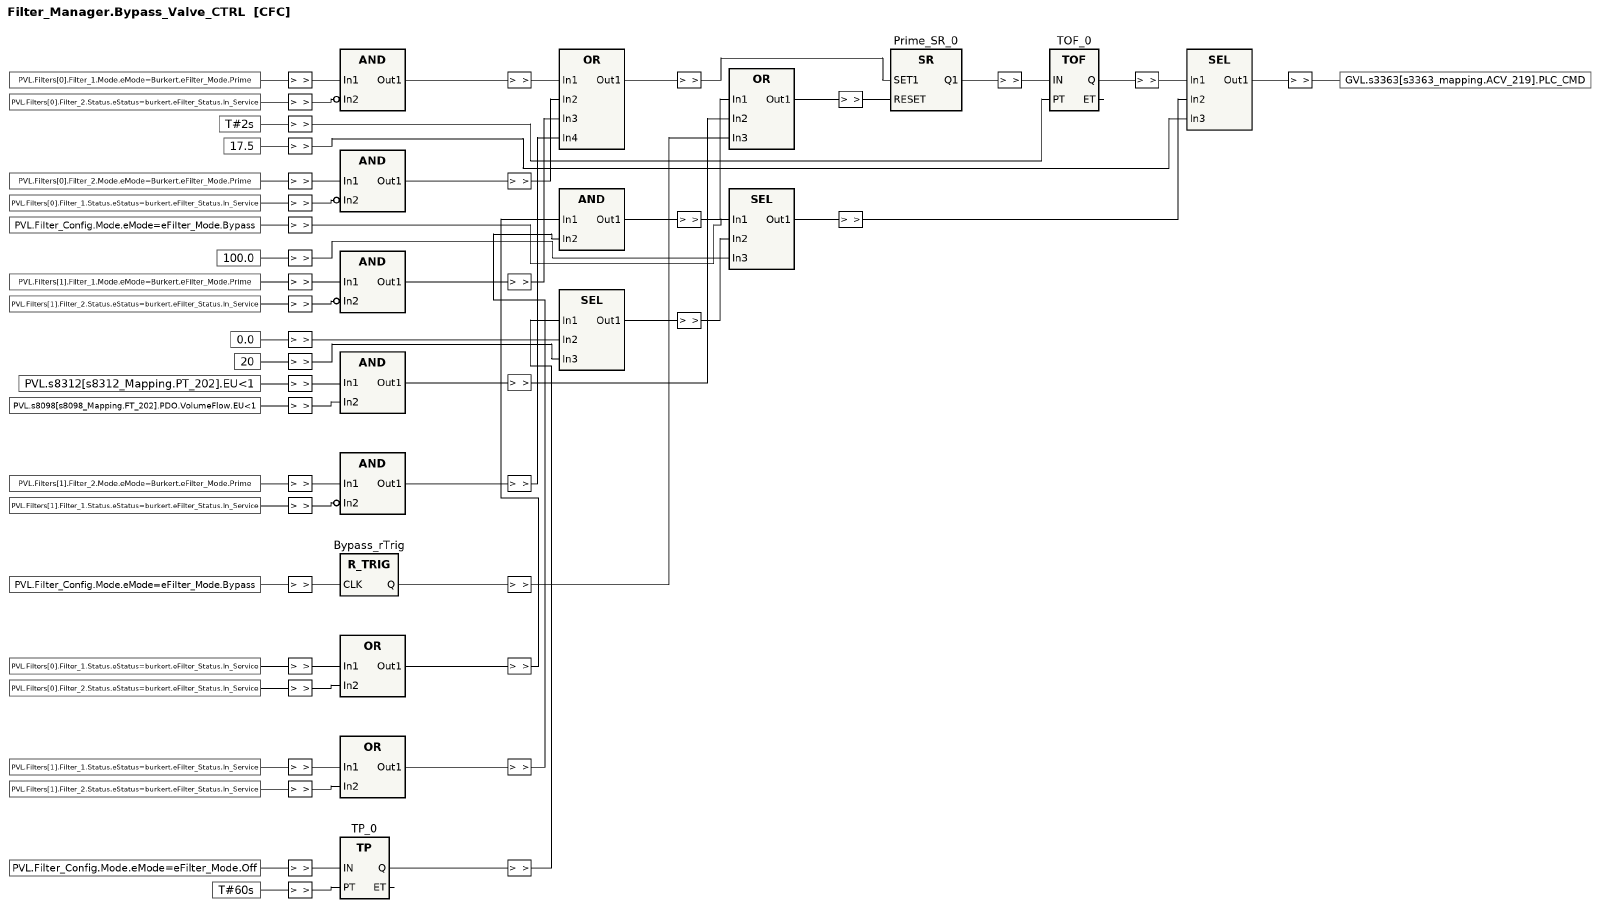
(* CFC diagram, written out as Structured Text *)
_OR8_OUT := (PVL.Filters[0].Filter_1.Status.eStatus=burkert.eFilter_Status.In_Service) OR (PVL.Filters[0].Filter_2.Status.eStatus=burkert.eFilter_Status.In_Service);
Prime_SR_0(SET1 := (PVL.Filters[0].Filter_1.Mode.eMode=Burkert.eFilter_Mode.Prime) AND NOT (PVL.Filters[0].Filter_2.Status.eStatus=burkert.eFilter_Status.In_Service) OR (PVL.Filters[0].Filter_2.Mode.eMode=Burkert.eFilter_Mode.Prime) AND NOT (PVL.Filters[0].Filter_1.Status.eStatus=burkert.eFilter_Status.In_Service) OR (PVL.Filters[1].Filter_1.Mode.eMode=Burkert.eFilter_Mode.Prime) AND NOT (PVL.Filters[1].Filter_2.Status.eStatus=burkert.eFilter_Status.In_Service) OR (PVL.Filters[1].Filter_2.Mode.eMode=Burkert.eFilter_Mode.Prime) AND NOT (PVL.Filters[1].Filter_1.Status.eStatus=burkert.eFilter_Status.In_Service), RESET := _OR43_OUT);
_SEL54_OUT_2 := SEL(TP_0.Q, 0.0, 20);
_OR43_OUT := _OR8_OUT AND ((PVL.Filters[1].Filter_1.Status.eStatus=burkert.eFilter_Status.In_Service) OR (PVL.Filters[1].Filter_2.Status.eStatus=burkert.eFilter_Status.In_Service)) OR _AND46_OUT OR Bypass_rTrig.Q;
_AND46_OUT := (PVL.s8312[s8312_Mapping.PT_202].EU<1) AND (PVL.s8098[s8098_Mapping.FT_202].PDO.VolumeFlow.EU<1);
TOF_0(IN := Prime_SR_0.Q1, PT := T#2s);
Bypass_rTrig(CLK := PVL.Filter_Config.Mode.eMode=eFilter_Mode.Bypass);
GVL.s3363[s3363_mapping.ACV_219].PLC_CMD := _SEL76_OUT;
_SEL76_OUT := SEL(TOF_0.Q, SEL(PVL.Filter_Config.Mode.eMode=eFilter_Mode.Bypass, _SEL54_OUT_2, 100.0), 17.5);
TP_0(IN := PVL.Filter_Config.Mode.eMode=eFilter_Mode.Off, PT := T#60s);
END_ACTION
END_PROGRAM

PROGRAM Correction
  VAR
    NaOCI_CND : Burkert.FB_LookUp_Table;
    NAOCI_X : ARRAY[0..19] OF REAL := [0, 3, 3.5, 4, 4.5, 5, 5.5];
    NaOCI_Y : ARRAY[0..19] OF REAL := [16.61, 101.9, 108.2, 116.2, 123.2, 133.8, 141.6];
    Test_X : REAL;
    Test_Y : REAL;
    Call_Query : BOOL;
  END_VAR

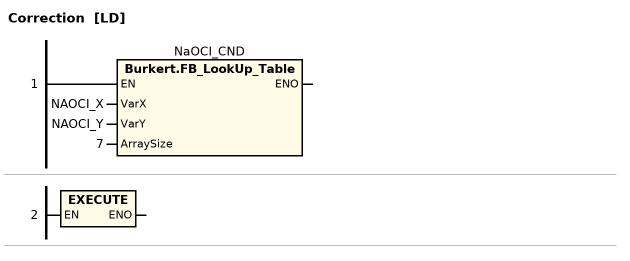
(* LD diagram, written out as Structured Text *)

NaOCI_CND(VarX := NAOCI_X, VarY := NAOCI_Y, ArraySize := 7);

IF Call_Query THEN
	Test_Y:=NaOCI_CND.GetVarY(InputX:=Test_X);
END_IF
END_PROGRAM

PROGRAM Level_0_CTRL

            //MEx3_ORF();
Stride_IO();

IoLink_Manager();
ME44_IO();
s8605_Manager();



          
END_PROGRAM

PROGRAM Z201_PWR
  VAR
    Override_Ton : Ton;
    StartUp_Complete : BOOL;
    RS_0 : RS;
    TP_0 : TP;
    TP_1 : TP;
    TP_2 : TP;
    TP_3 : TP;
    TON_0 : TON;
    TP_4 : TP;
    TON_1 : TON;
    TON_2 : TON;
    TON_3 : TON;
  END_VAR
  VAR  (* added by the conversion: wires and edge detectors of the diagram *)
    _AND3_OUT : BOOL;
    _OR21_OUT : BOOL;
    _AND27_OUT : BOOL;
    _AND49_OUT : BOOL;
    _OR43_OUT : BOOL;
    _AND72_OUT : BOOL;
    _OR66_OUT : BOOL;
    _AND95_OUT : BOOL;
    _OR89_OUT : BOOL;
    _AND129_OUT : BOOL;
    _MOVE144_ENO : BOOL;
    _MOVE144_OUT : BOOL;
  END_VAR

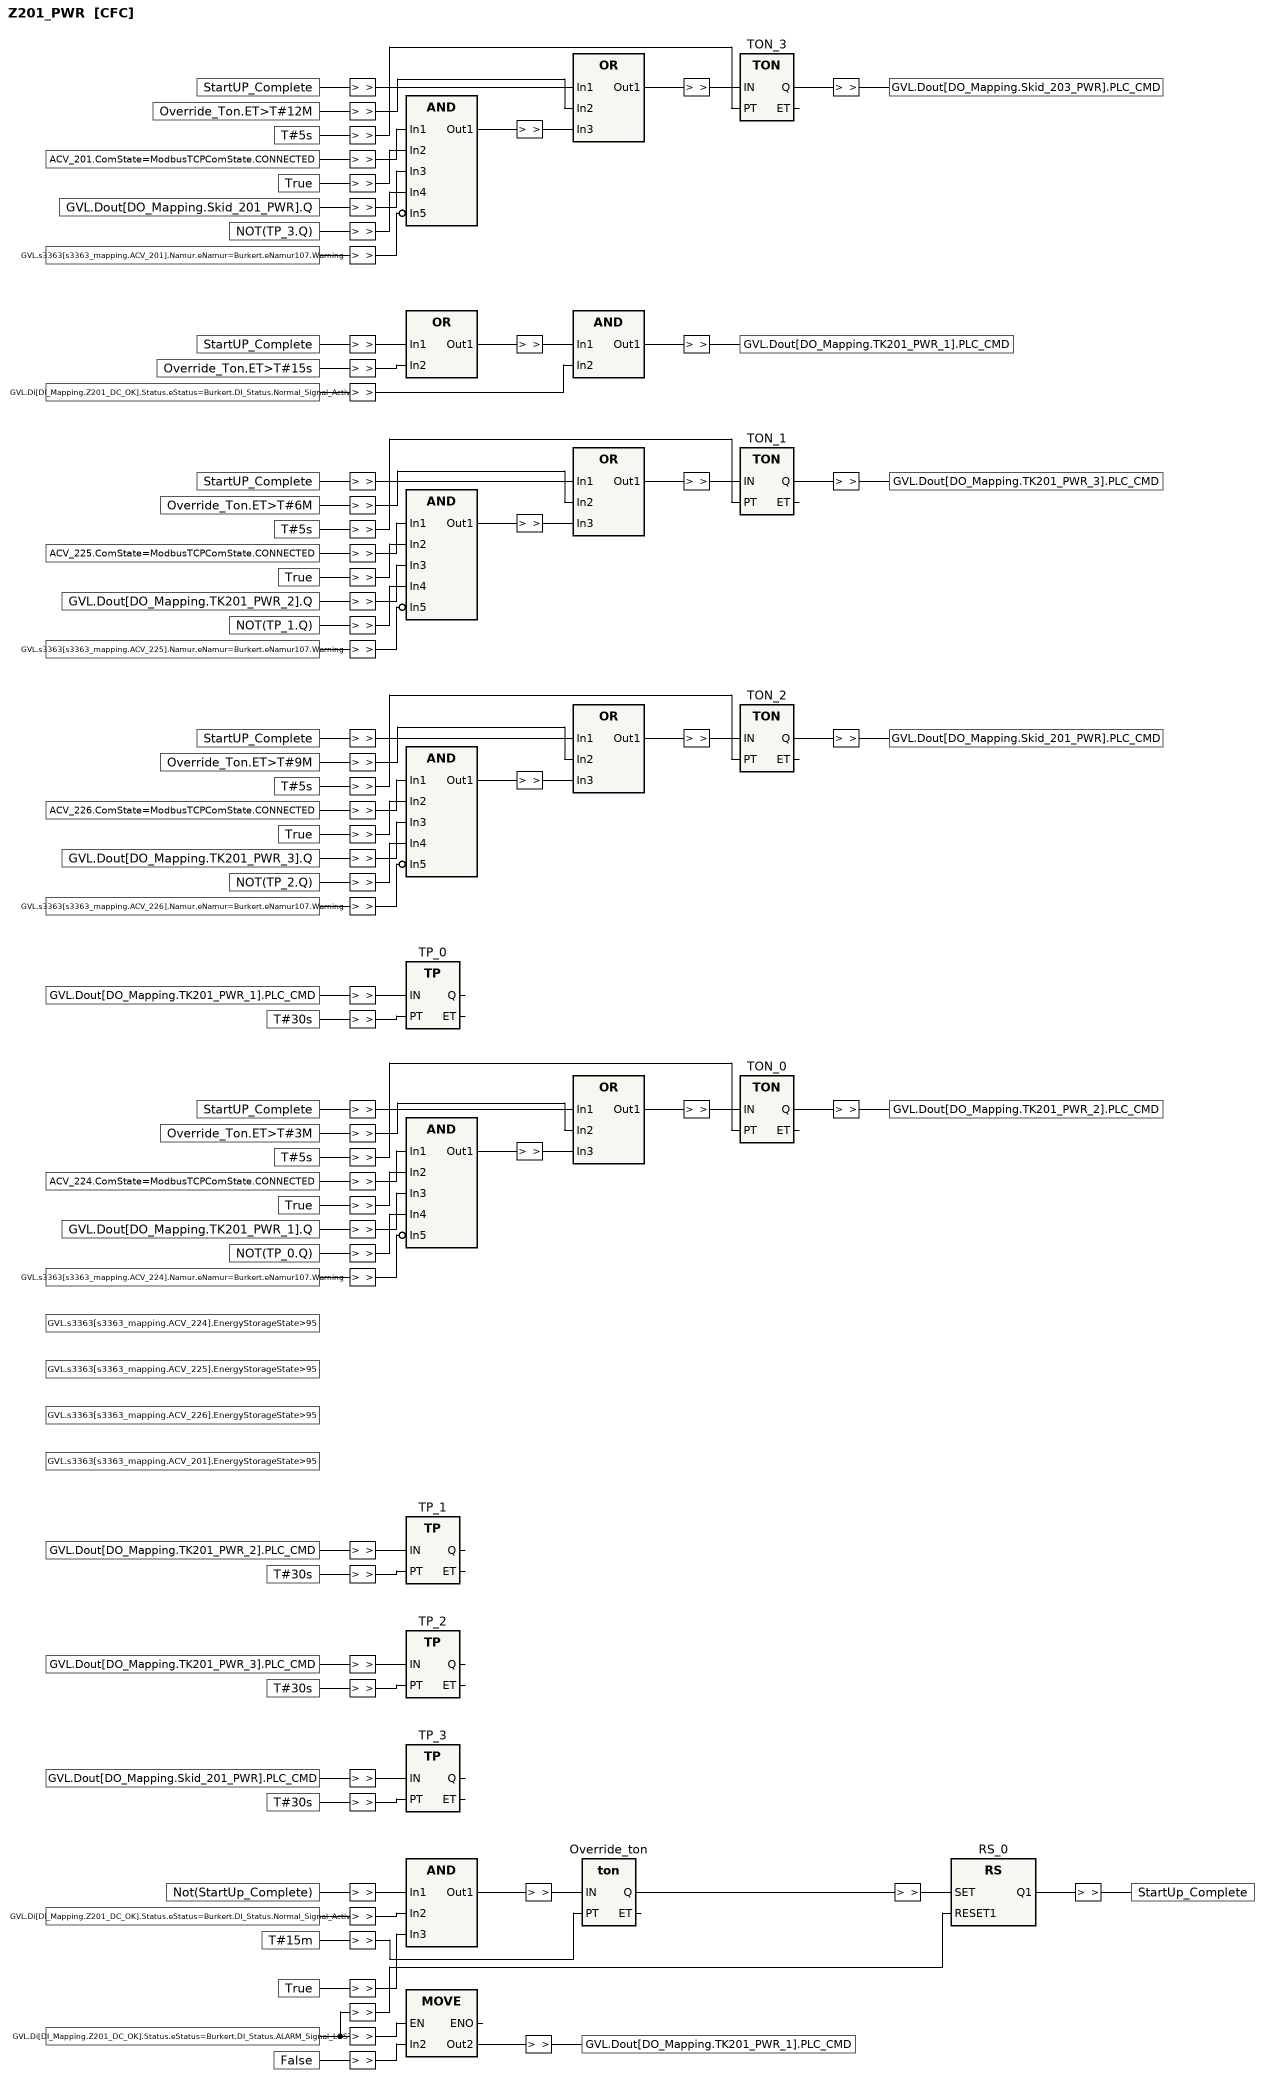
(* CFC diagram, written out as Structured Text *)
GVL.Dout[DO_Mapping.TK201_PWR_1].PLC_CMD := _AND3_OUT;
TP_0(IN := GVL.Dout[DO_Mapping.TK201_PWR_1].PLC_CMD, PT := T#30s);
TON_0(IN := _OR21_OUT, PT := T#5s);
_OR21_OUT := StartUP_Complete OR (Override_Ton.ET>T#3M) OR _AND27_OUT;
GVL.Dout[DO_Mapping.TK201_PWR_2].PLC_CMD := TON_0.Q;
_OR43_OUT := StartUP_Complete OR (Override_Ton.ET>T#6M) OR _AND49_OUT;
GVL.Dout[DO_Mapping.TK201_PWR_3].PLC_CMD := TON_1.Q;
_AND49_OUT := (ACV_225.ComState=ModbusTCPComState.CONNECTED) AND True AND GVL.Dout[DO_Mapping.TK201_PWR_2].Q AND NOT(TP_1.Q) AND NOT (GVL.s3363[s3363_mapping.ACV_225].Namur.eNamur=Burkert.eNamur107.Warning);
_OR66_OUT := StartUP_Complete OR (Override_Ton.ET>T#9M) OR _AND72_OUT;
GVL.Dout[DO_Mapping.Skid_201_PWR].PLC_CMD := TON_2.Q;
_AND72_OUT := (ACV_226.ComState=ModbusTCPComState.CONNECTED) AND True AND GVL.Dout[DO_Mapping.TK201_PWR_3].Q AND NOT(TP_2.Q) AND NOT (GVL.s3363[s3363_mapping.ACV_226].Namur.eNamur=Burkert.eNamur107.Warning);
_OR89_OUT := StartUP_Complete OR (Override_Ton.ET>T#12M) OR _AND95_OUT;
GVL.Dout[DO_Mapping.Skid_203_PWR].PLC_CMD := TON_3.Q;
_AND95_OUT := (ACV_201.ComState=ModbusTCPComState.CONNECTED) AND True AND GVL.Dout[DO_Mapping.Skid_201_PWR].Q AND NOT(TP_3.Q) AND NOT (GVL.s3363[s3363_mapping.ACV_201].Namur.eNamur=Burkert.eNamur107.Warning);
TP_1(IN := GVL.Dout[DO_Mapping.TK201_PWR_2].PLC_CMD, PT := T#30s);
TP_2(IN := GVL.Dout[DO_Mapping.TK201_PWR_3].PLC_CMD, PT := T#30s);
TP_3(IN := GVL.Dout[DO_Mapping.Skid_201_PWR].PLC_CMD, PT := T#30s);
Override_ton(IN := _AND129_OUT, PT := T#15m);
RS_0(SET := Override_ton.Q, RESET1 := GVL.Di[DI_Mapping.Z201_DC_OK].Status.eStatus=Burkert.DI_Status.ALARM_Signal_LOST);
_AND129_OUT := Not(StartUp_Complete) AND (GVL.Di[DI_Mapping.Z201_DC_OK].Status.eStatus=Burkert.DI_Status.Normal_Signal_Active) AND True;
StartUp_Complete := RS_0.Q1;
_MOVE144_OUT := MOVE(EN := GVL.Di[DI_Mapping.Z201_DC_OK].Status.eStatus=Burkert.DI_Status.ALARM_Signal_LOST, IN := False, ENO => _MOVE144_ENO);
IF _MOVE144_ENO THEN GVL.Dout[DO_Mapping.TK201_PWR_1].PLC_CMD := _MOVE144_OUT; END_IF;
TON_3(IN := _OR89_OUT, PT := T#5s);
TON_1(IN := _OR43_OUT, PT := T#5s);
TON_2(IN := _OR66_OUT, PT := T#5s);
_AND3_OUT := (StartUP_Complete OR (Override_Ton.ET>T#15s)) AND (GVL.Di[DI_Mapping.Z201_DC_OK].Status.eStatus=Burkert.DI_Status.Normal_Signal_Active);
_AND27_OUT := (ACV_224.ComState=ModbusTCPComState.CONNECTED) AND True AND GVL.Dout[DO_Mapping.TK201_PWR_1].Q AND NOT(TP_0.Q) AND NOT (GVL.s3363[s3363_mapping.ACV_224].Namur.eNamur=Burkert.eNamur107.Warning);
(* drawn but not wired to any output: GVL.s3363[s3363_mapping.ACV_224].EnergyStorageState>95, GVL.s3363[s3363_mapping.ACV_225].EnergyStorageState>95, GVL.s3363[s3363_mapping.ACV_226].EnergyStorageState>95, GVL.s3363[s3363_mapping.ACV_201].EnergyStorageState>95 *)
END_PROGRAM

PROGRAM IoLink_Manager
  VAR
    Z201_GW : Burkert.AL1340_UDFB;
    Z202_GW : Burkert.AL1340_UDFB;
  END_VAR

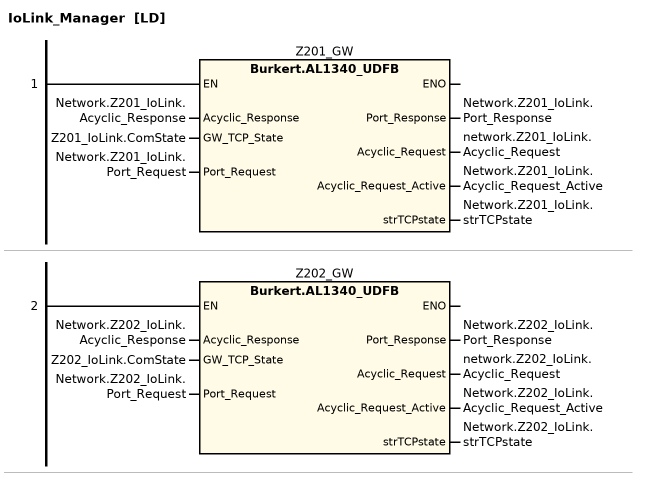
(* LD diagram, written out as Structured Text *)

Z201_GW(Acyclic_Response := Network.Z201_IoLink.Acyclic_Response, GW_TCP_State := Z201_IoLink.ComState, Port_Request := Network.Z201_IoLink.Port_Request, Port_Response => Network.Z201_IoLink.Port_Response, Acyclic_Request => network.Z201_IoLink.Acyclic_Request, Acyclic_Request_Active => Network.Z201_IoLink.Acyclic_Request_Active, strTCPstate => Network.Z201_IoLink.strTCPstate);

Z202_GW(Acyclic_Response := Network.Z202_IoLink.Acyclic_Response, GW_TCP_State := Z202_IoLink.ComState, Port_Request := Network.Z202_IoLink.Port_Request, Port_Response => Network.Z202_IoLink.Port_Response, Acyclic_Request => network.Z202_IoLink.Acyclic_Request, Acyclic_Request_Active => Network.Z202_IoLink.Acyclic_Request_Active, strTCPstate => Network.Z202_IoLink.strTCPstate);
(* --- network --- *)
END_PROGRAM

PROGRAM Flowave_Manager
  VAR
    FT_101_CTRL : Burkert.eDip_8098_CTRL;
    FT_201_CTRL : Burkert.eDip_8098_CTRL;
    FT_202_CTRL : Burkert.eDip_8098_CTRL;
    FT_203_CTRL : Burkert.eDip_8098_CTRL;
    FT_204_CTRL : Burkert.eDip_8098_CTRL;
  END_VAR

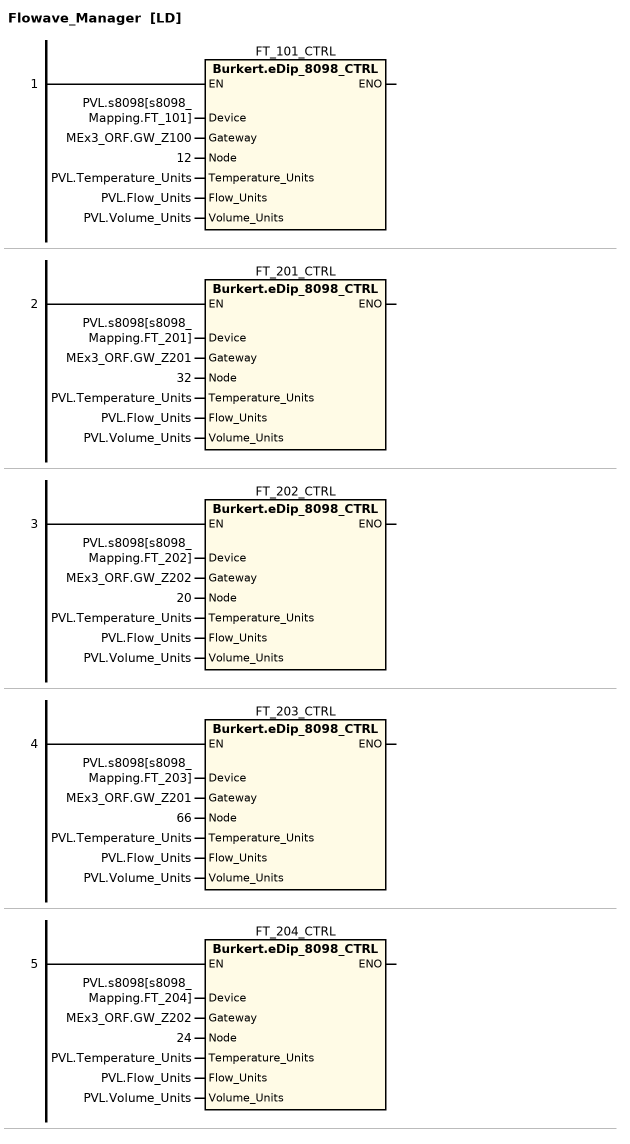
(* LD diagram, written out as Structured Text *)

FT_101_CTRL(Device := PVL.s8098[s8098_Mapping.FT_101], Gateway := MEx3_ORF.GW_Z100, Node := 12, Temperature_Units := PVL.Temperature_Units, Flow_Units := PVL.Flow_Units, Volume_Units := PVL.Volume_Units);

FT_201_CTRL(Device := PVL.s8098[s8098_Mapping.FT_201], Gateway := MEx3_ORF.GW_Z201, Node := 32, Temperature_Units := PVL.Temperature_Units, Flow_Units := PVL.Flow_Units, Volume_Units := PVL.Volume_Units);

FT_202_CTRL(Device := PVL.s8098[s8098_Mapping.FT_202], Gateway := MEx3_ORF.GW_Z202, Node := 20, Temperature_Units := PVL.Temperature_Units, Flow_Units := PVL.Flow_Units, Volume_Units := PVL.Volume_Units);

FT_203_CTRL(Device := PVL.s8098[s8098_Mapping.FT_203], Gateway := MEx3_ORF.GW_Z201, Node := 66, Temperature_Units := PVL.Temperature_Units, Flow_Units := PVL.Flow_Units, Volume_Units := PVL.Volume_Units);

FT_204_CTRL(Device := PVL.s8098[s8098_Mapping.FT_204], Gateway := MEx3_ORF.GW_Z202, Node := 24, Temperature_Units := PVL.Temperature_Units, Flow_Units := PVL.Flow_Units, Volume_Units := PVL.Volume_Units);
END_PROGRAM

PROGRAM Z202_PWR
  VAR
    Override_Ton : Ton;
    StartUp_Complete : BOOL;
    RS_0 : RS;
    Master_Off : BOOL;
    TP_0 : TP;
    TP_1 : TP;
    TP_2 : TP;
    TP_3 : TP;
    TON_0 : Ton;
    TON_1 : Ton;
    TON_2 : Ton;
    TON_3 : Ton;
    TON_4 : TON;
    TON_5 : TON;
    TON_6 : TON;
    TON_7 : TON;
  END_VAR
  VAR  (* added by the conversion: wires and edge detectors of the diagram *)
    _AND0_OUT : BOOL;
    _MOVE13_OUT : ANY;
    _AND115_OUT : BOOL;
    _OR111_OUT : BOOL;
    _AND155_OUT : BOOL;
    _OR168_OUT : BOOL;
    _OR179_OUT : BOOL;
    _AND177_OUT : BOOL;
    _MOVE190_ENO : BOOL;
    _MOVE190_OUT : BOOL;
    _SEL45_OUT : ANY;
    _OR202_OUT : BOOL;
    _AND68_OUT : BOOL;
    _MOVE13_ENO : BOOL;
  END_VAR

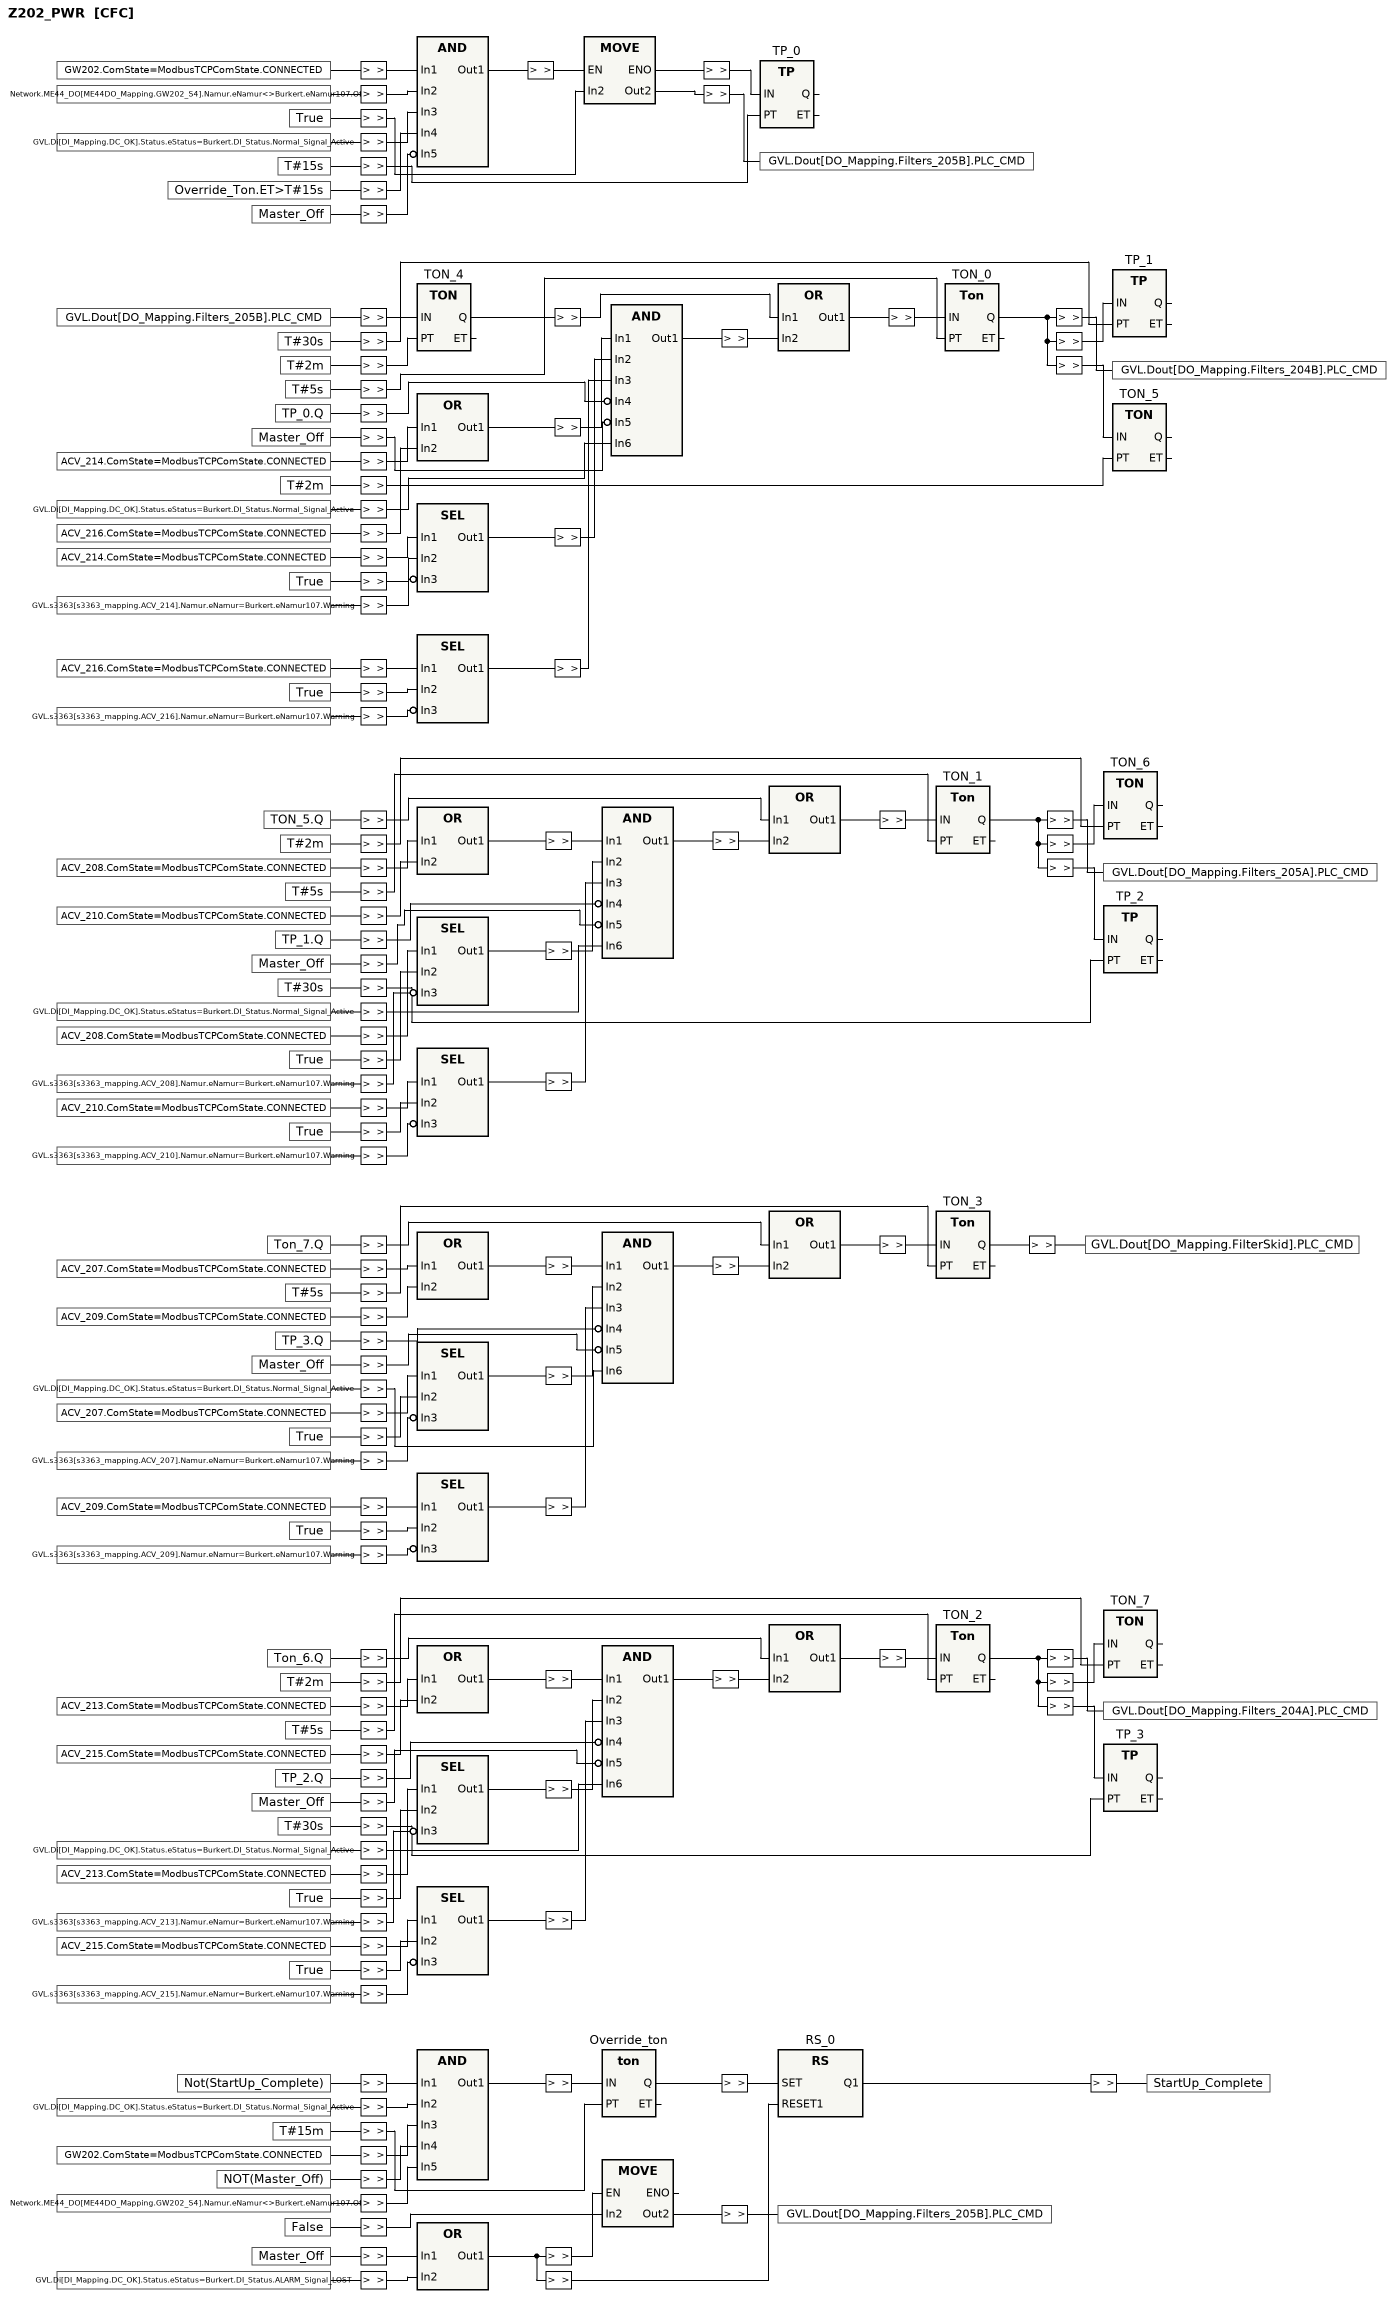
(* CFC diagram, written out as Structured Text *)
_AND0_OUT := (GW202.ComState=ModbusTCPComState.CONNECTED) AND (Network.ME44_DO[ME44DO_Mapping.GW202_S4].Namur.eNamur<>Burkert.eNamur107.Offline) AND (GVL.Di[DI_Mapping.DC_OK].Status.eStatus=Burkert.DI_Status.Normal_Signal_Active) AND (Override_Ton.ET>T#15s) AND NOT Master_Off;
GVL.Dout[DO_Mapping.Filters_205B].PLC_CMD := _MOVE13_OUT;
TON_4(IN := GVL.Dout[DO_Mapping.Filters_205B].PLC_CMD, PT := T#2m);
GVL.Dout[DO_Mapping.Filters_204B].PLC_CMD := TON_0.Q;
GVL.Dout[DO_Mapping.Filters_205A].PLC_CMD := TON_1.Q;
TP_0(IN := _MOVE13_OUT, PT := T#15s);
_OR111_OUT := Ton_6.Q OR _AND115_OUT;
GVL.Dout[DO_Mapping.Filters_204A].PLC_CMD := TON_2.Q;
_AND155_OUT := Not(StartUp_Complete) AND (GVL.Di[DI_Mapping.DC_OK].Status.eStatus=Burkert.DI_Status.Normal_Signal_Active) AND (GW202.ComState=ModbusTCPComState.CONNECTED) AND NOT(Master_Off) AND (Network.ME44_DO[ME44DO_Mapping.GW202_S4].Namur.eNamur<>Burkert.eNamur107.Offline);
_OR168_OUT := Master_Off OR (GVL.Di[DI_Mapping.DC_OK].Status.eStatus=Burkert.DI_Status.ALARM_Signal_LOST);
_AND177_OUT := _OR179_OUT AND SEL(ACV_207.ComState=ModbusTCPComState.CONNECTED, True, NOT (GVL.s3363[s3363_mapping.ACV_207].Namur.eNamur=Burkert.eNamur107.Warning)) AND SEL(ACV_209.ComState=ModbusTCPComState.CONNECTED, True, NOT (GVL.s3363[s3363_mapping.ACV_209].Namur.eNamur=Burkert.eNamur107.Warning)) AND NOT TP_3.Q AND NOT Master_Off AND (GVL.Di[DI_Mapping.DC_OK].Status.eStatus=Burkert.DI_Status.Normal_Signal_Active);
_MOVE190_OUT := MOVE(EN := _OR168_OUT, IN := False, ENO => _MOVE190_ENO);
IF _MOVE190_ENO THEN GVL.Dout[DO_Mapping.Filters_205B].PLC_CMD := _MOVE190_OUT; END_IF;
_SEL45_OUT := SEL(ACV_216.ComState=ModbusTCPComState.CONNECTED, True, NOT (GVL.s3363[s3363_mapping.ACV_216].Namur.eNamur=Burkert.eNamur107.Warning));
TP_1(IN := TON_0.Q, PT := T#30s);
TON_0(IN := TON_4.Q OR ((ACV_214.ComState=ModbusTCPComState.CONNECTED) OR (ACV_216.ComState=ModbusTCPComState.CONNECTED)) AND SEL(ACV_214.ComState=ModbusTCPComState.CONNECTED, True, NOT (GVL.s3363[s3363_mapping.ACV_214].Namur.eNamur=Burkert.eNamur107.Warning)) AND _SEL45_OUT AND NOT TP_0.Q AND NOT Master_Off AND (GVL.Di[DI_Mapping.DC_OK].Status.eStatus=Burkert.DI_Status.Normal_Signal_Active), PT := T#5s);
TON_3(IN := _OR202_OUT, PT := T#5s);
TON_5(IN := TON_0.Q, PT := T#2m);
TON_6(IN := TON_1.Q, PT := T#2m);
TP_2(IN := TON_1.Q, PT := T#30s);
TON_7(IN := TON_2.Q, PT := T#2m);
TP_3(IN := TON_2.Q, PT := T#30s);
TON_1(IN := TON_5.Q OR _AND68_OUT, PT := T#5s);
TON_2(IN := _OR111_OUT, PT := T#5s);
RS_0(SET := Override_ton.Q, RESET1 := _OR168_OUT);
Override_ton(IN := _AND155_OUT, PT := T#15m);
GVL.Dout[DO_Mapping.FilterSkid].PLC_CMD := TON_3.Q;
_AND68_OUT := ((ACV_208.ComState=ModbusTCPComState.CONNECTED) OR (ACV_210.ComState=ModbusTCPComState.CONNECTED)) AND SEL(ACV_208.ComState=ModbusTCPComState.CONNECTED, True, NOT (GVL.s3363[s3363_mapping.ACV_208].Namur.eNamur=Burkert.eNamur107.Warning)) AND SEL(ACV_210.ComState=ModbusTCPComState.CONNECTED, True, NOT (GVL.s3363[s3363_mapping.ACV_210].Namur.eNamur=Burkert.eNamur107.Warning)) AND NOT TP_1.Q AND NOT Master_Off AND (GVL.Di[DI_Mapping.DC_OK].Status.eStatus=Burkert.DI_Status.Normal_Signal_Active);
_AND115_OUT := ((ACV_213.ComState=ModbusTCPComState.CONNECTED) OR (ACV_215.ComState=ModbusTCPComState.CONNECTED)) AND SEL(ACV_213.ComState=ModbusTCPComState.CONNECTED, True, NOT (GVL.s3363[s3363_mapping.ACV_213].Namur.eNamur=Burkert.eNamur107.Warning)) AND SEL(ACV_215.ComState=ModbusTCPComState.CONNECTED, True, NOT (GVL.s3363[s3363_mapping.ACV_215].Namur.eNamur=Burkert.eNamur107.Warning)) AND NOT TP_2.Q AND NOT Master_Off AND (GVL.Di[DI_Mapping.DC_OK].Status.eStatus=Burkert.DI_Status.Normal_Signal_Active);
_OR202_OUT := Ton_7.Q OR _AND177_OUT;
_OR179_OUT := (ACV_207.ComState=ModbusTCPComState.CONNECTED) OR (ACV_209.ComState=ModbusTCPComState.CONNECTED);
StartUp_Complete := RS_0.Q1;
_MOVE13_OUT := MOVE(EN := _AND0_OUT, IN := True, ENO => _MOVE13_ENO);
END_PROGRAM

PROGRAM BCV_Manager
  VAR
    BCV_211_CTRL : Burkert.Basic_BCV_UDFB;
    BCV_212_CTRL : Burkert.Basic_BCV_UDFB;
    BCV_217_CTRL : Burkert.Basic_BCV_UDFB;
    BCV_218_CTRL : Burkert.Basic_BCV_UDFB;
    BCV_220_CTRL : Burkert.Basic_BCV_UDFB;
    BCV_221_CTRL : Burkert.Basic_BCV_UDFB;
    BCV_222_CTRL : Burkert.Basic_BCV_UDFB;
    BCV_223_CTRL : Burkert.Basic_BCV_UDFB;
  END_VAR

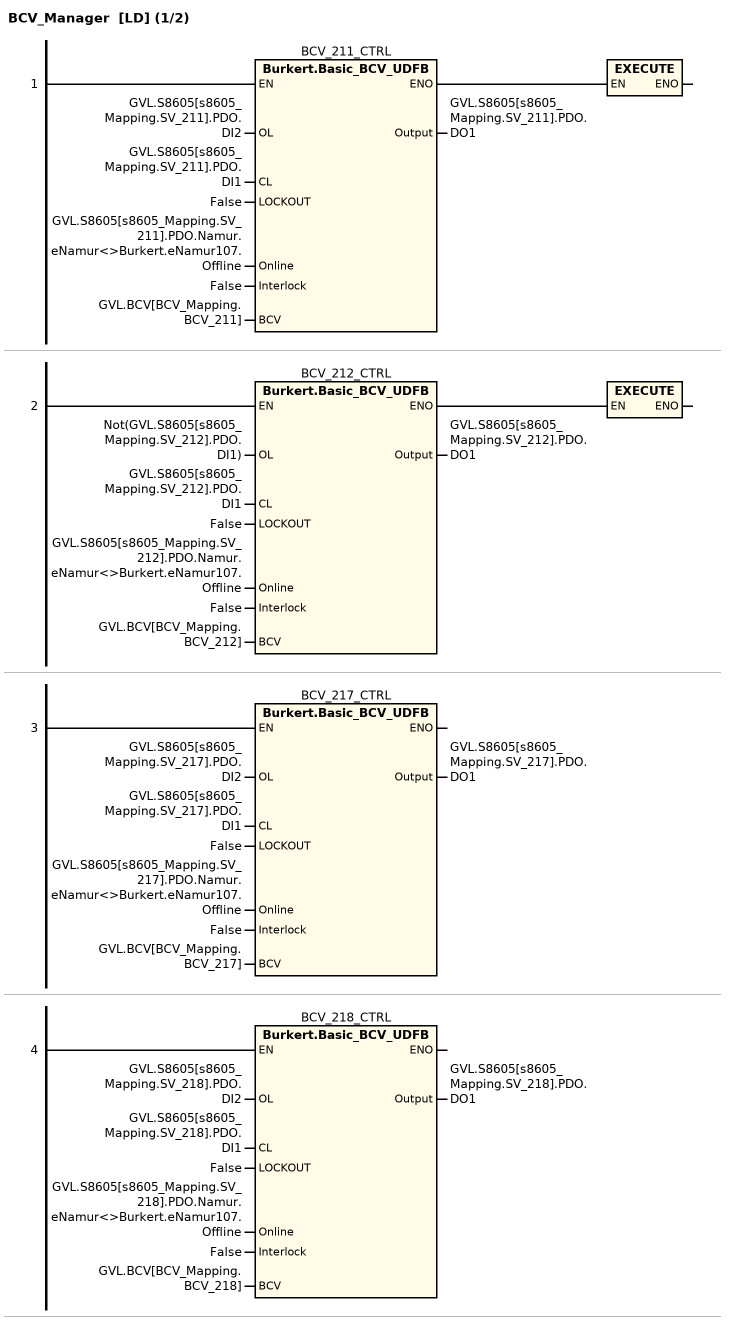
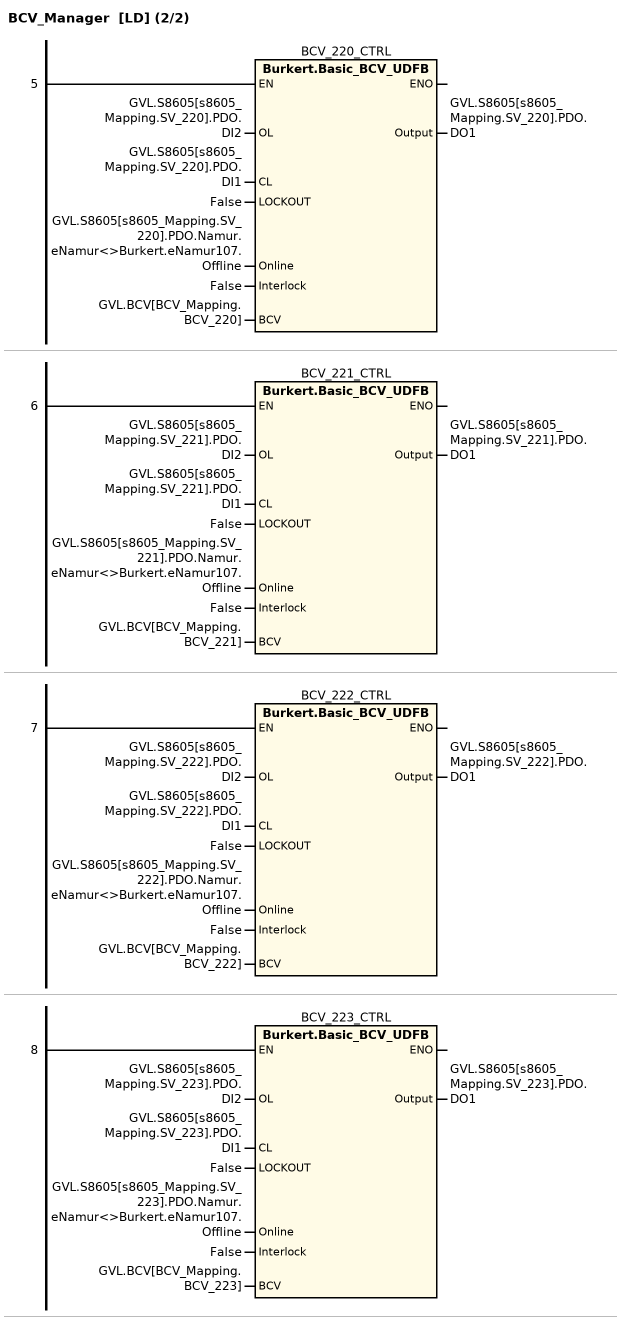
(* LD diagram, written out as Structured Text *)

BCV_211_CTRL(OL := GVL.S8605[s8605_Mapping.SV_211].PDO.DI2, CL := GVL.S8605[s8605_Mapping.SV_211].PDO.DI1, LOCKOUT := False, Online := GVL.S8605[s8605_Mapping.SV_211].PDO.Namur.eNamur<>Burkert.eNamur107.Offline, Interlock := False, BCV := GVL.BCV[BCV_Mapping.BCV_211], Output => GVL.S8605[s8605_Mapping.SV_211].PDO.DO1);
IF BCV_211_CTRL.ENO THEN
  //GVL.S8605[s8605_Mapping.SV_211].PDO.DI2
END_IF;

BCV_212_CTRL(OL := Not(GVL.S8605[s8605_Mapping.SV_212].PDO.DI1), CL := GVL.S8605[s8605_Mapping.SV_212].PDO.DI1, LOCKOUT := False, Online := GVL.S8605[s8605_Mapping.SV_212].PDO.Namur.eNamur<>Burkert.eNamur107.Offline, Interlock := False, BCV := GVL.BCV[BCV_Mapping.BCV_212], Output => GVL.S8605[s8605_Mapping.SV_212].PDO.DO1);
IF BCV_212_CTRL.ENO THEN
  //GVL.S8605[s8605_Mapping.SV_212].PDO.DI2
END_IF;

BCV_217_CTRL(OL := GVL.S8605[s8605_Mapping.SV_217].PDO.DI2, CL := GVL.S8605[s8605_Mapping.SV_217].PDO.DI1, LOCKOUT := False, Online := GVL.S8605[s8605_Mapping.SV_217].PDO.Namur.eNamur<>Burkert.eNamur107.Offline, Interlock := False, BCV := GVL.BCV[BCV_Mapping.BCV_217], Output => GVL.S8605[s8605_Mapping.SV_217].PDO.DO1);

BCV_218_CTRL(OL := GVL.S8605[s8605_Mapping.SV_218].PDO.DI2, CL := GVL.S8605[s8605_Mapping.SV_218].PDO.DI1, LOCKOUT := False, Online := GVL.S8605[s8605_Mapping.SV_218].PDO.Namur.eNamur<>Burkert.eNamur107.Offline, Interlock := False, BCV := GVL.BCV[BCV_Mapping.BCV_218], Output => GVL.S8605[s8605_Mapping.SV_218].PDO.DO1);

BCV_220_CTRL(OL := GVL.S8605[s8605_Mapping.SV_220].PDO.DI2, CL := GVL.S8605[s8605_Mapping.SV_220].PDO.DI1, LOCKOUT := False, Online := GVL.S8605[s8605_Mapping.SV_220].PDO.Namur.eNamur<>Burkert.eNamur107.Offline, Interlock := False, BCV := GVL.BCV[BCV_Mapping.BCV_220], Output => GVL.S8605[s8605_Mapping.SV_220].PDO.DO1);

BCV_221_CTRL(OL := GVL.S8605[s8605_Mapping.SV_221].PDO.DI2, CL := GVL.S8605[s8605_Mapping.SV_221].PDO.DI1, LOCKOUT := False, Online := GVL.S8605[s8605_Mapping.SV_221].PDO.Namur.eNamur<>Burkert.eNamur107.Offline, Interlock := False, BCV := GVL.BCV[BCV_Mapping.BCV_221], Output => GVL.S8605[s8605_Mapping.SV_221].PDO.DO1);

